// TIA Portal V20 export
DATA_BLOCK "ST_INPUT_Map_DB"   // DB102
{ S7_Optimized_Access := 'FALSE' }
// stored: AutoNumber false
   VAR
      "I0.0" { ExternalVisible := 'False'} : Bool := FALSE;   // I0.0
      "I0.1" { ExternalVisible := 'False'} : Bool := FALSE;   // I0.1
      "I0.2" { ExternalVisible := 'False'} : Bool := FALSE;   // I0.2
      "I0.3" { ExternalVisible := 'False'} : Bool := FALSE;   // I0.3
      "I0.4" { ExternalVisible := 'False'} : Bool := FALSE;   // I0.4
      "I0.5" { ExternalVisible := 'False'} : Bool := FALSE;   // I0.5
      "I0.6" { ExternalVisible := 'False'} : Bool := FALSE;   // I0.6
      "I0.7" { ExternalVisible := 'False'} : Bool := FALSE;   // I0.7
      "I1.0" { ExternalVisible := 'False'} : Bool := FALSE;   // I1.0
      "I1.1" { ExternalVisible := 'False'} : Bool := FALSE;   // I1.1
      "I1.2" { ExternalVisible := 'False'} : Bool := FALSE;   // I1.2
      "I1.3" { ExternalVisible := 'False'} : Bool := FALSE;   // I1.3
      "I1.4" { ExternalVisible := 'False'} : Bool := FALSE;   // I1.4
      "I1.5" { ExternalVisible := 'False'} : Bool := FALSE;   // I1.5
      "I1.6" { ExternalVisible := 'False'} : Bool := FALSE;   // I1.6
      "I1.7" { ExternalVisible := 'False'} : Bool := FALSE;   // I1.7
      "I2.0" { ExternalVisible := 'False'} : Bool := FALSE;   // I2.0
      "I2.1" { ExternalVisible := 'False'} : Bool := FALSE;   // I2.1
      "I2.2" { ExternalVisible := 'False'} : Bool := FALSE;   // I2.2
      "I2.3" { ExternalVisible := 'False'} : Bool := FALSE;   // I2.3
      "I2.4" { ExternalVisible := 'False'} : Bool := FALSE;   // I2.4
      "I2.5" { ExternalVisible := 'False'} : Bool := FALSE;   // I2.5
      "I2.6" { ExternalVisible := 'False'} : Bool := FALSE;   // I2.6
      "I2.7" { ExternalVisible := 'False'} : Bool := FALSE;   // I2.7
      "I3.0" { ExternalVisible := 'False'} : Bool := FALSE;   // I3.0
      "I3.1" { ExternalVisible := 'False'} : Bool := FALSE;   // I3.1
      "I3.2" { ExternalVisible := 'False'} : Bool := FALSE;   // I3.2
      "I3.3" { ExternalVisible := 'False'} : Bool := FALSE;   // I3.3
      "I3.4" { ExternalVisible := 'False'} : Bool := FALSE;   // I3.4
      "I3.5" { ExternalVisible := 'False'} : Bool := FALSE;   // I3.5
      "I3.6" { ExternalVisible := 'False'} : Bool := FALSE;   // I3.6
      "I3.7" { ExternalVisible := 'False'} : Bool := FALSE;   // I3.7
      "I4.0" { ExternalVisible := 'False'} : Bool := FALSE;   // I4.0
      "I4.1" { ExternalVisible := 'False'} : Bool := FALSE;   // I4.1
      "I4.2" { ExternalVisible := 'False'} : Bool := FALSE;   // I4.2
      "I4.3" { ExternalVisible := 'False'} : Bool := FALSE;   // I4.3
      "I4.4" { ExternalVisible := 'False'} : Bool := FALSE;   // I4.4
      "I4.5" { ExternalVisible := 'False'} : Bool := FALSE;   // I4.5
      "I4.6" { ExternalVisible := 'False'} : Bool := FALSE;   // I4.6
      "I4.7" { ExternalVisible := 'False'} : Bool := FALSE;   // I4.7
      "I5.0" { ExternalVisible := 'False'} : Bool := FALSE;   // I5.0
      "I5.1" { ExternalVisible := 'False'} : Bool := FALSE;   // I5.1
      "I5.2" { ExternalVisible := 'False'} : Bool := FALSE;   // I5.2
      "I5.3" { ExternalVisible := 'False'} : Bool := FALSE;   // I5.3
      "I5.4" { ExternalVisible := 'False'} : Bool := FALSE;   // I5.4
      "I5.5" { ExternalVisible := 'False'} : Bool := FALSE;   // I5.5
      "I5.6" { ExternalVisible := 'False'} : Bool := FALSE;   // I5.6
      "I5.7" { ExternalVisible := 'False'} : Bool := FALSE;   // I5.7
      "I6.0" { ExternalVisible := 'False'} : Bool := FALSE;   // I6.0
      "I6.1" { ExternalVisible := 'False'} : Bool := FALSE;   // I6.1
      "I6.2" { ExternalVisible := 'False'} : Bool := FALSE;   // I6.2
      "I6.3" { ExternalVisible := 'False'} : Bool := FALSE;   // I6.3
      "I6.4" { ExternalVisible := 'False'} : Bool := FALSE;   // I6.4
      "I6.5" { ExternalVisible := 'False'} : Bool := FALSE;   // I6.5
      "I6.6" { ExternalVisible := 'False'} : Bool := FALSE;   // I6.6
      "I6.7" { ExternalVisible := 'False'} : Bool := FALSE;   // I6.7
      "I7.0" { ExternalVisible := 'False'} : Bool := FALSE;   // I7.0
      "I7.1" { ExternalVisible := 'False'} : Bool := FALSE;   // I7.1
      "I7.2" { ExternalVisible := 'False'} : Bool := FALSE;   // I7.2
      "I7.3" { ExternalVisible := 'False'} : Bool := FALSE;   // I7.3
      "I7.4" { ExternalVisible := 'False'} : Bool := FALSE;   // I7.4
      "I7.5" { ExternalVisible := 'False'} : Bool := FALSE;   // I7.5
      "I7.6" { ExternalVisible := 'False'} : Bool := FALSE;   // I7.6
      "I7.7" { ExternalVisible := 'False'} : Bool := FALSE;   // I7.7
      "I8.0" { ExternalVisible := 'False'} : Bool := FALSE;   // I8.0
      "I8.1" { ExternalVisible := 'False'} : Bool := FALSE;   // I8.1
      "I8.2" { ExternalVisible := 'False'} : Bool := FALSE;   // I8.2
      "I8.3" { ExternalVisible := 'False'} : Bool := FALSE;   // I8.3
      "I8.4" { ExternalVisible := 'False'} : Bool := FALSE;   // I8.4
      "I8.5" { ExternalVisible := 'False'} : Bool := FALSE;   // I8.5
      "I8.6" { ExternalVisible := 'False'} : Bool := FALSE;   // I8.6
      "I8.7" { ExternalVisible := 'False'} : Bool := FALSE;   // I8.7
      "I9.0" { ExternalVisible := 'False'} : Bool := FALSE;   // I9.0
      "I9.1" { ExternalVisible := 'False'} : Bool := FALSE;   // I9.1
      "I9.2" { ExternalVisible := 'False'} : Bool := FALSE;   // I9.2
      "I9.3" { ExternalVisible := 'False'} : Bool := FALSE;   // I9.3
      "I9.4" { ExternalVisible := 'False'} : Bool := FALSE;   // I9.4
      "I9.5" { ExternalVisible := 'False'} : Bool := FALSE;   // I9.5
      "I9.6" { ExternalVisible := 'False'} : Bool := FALSE;   // I9.6
      "I9.7" { ExternalVisible := 'False'} : Bool := FALSE;   // I9.7
      F31 { ExternalVisible := 'False'} : Bool := FALSE;   // HMI供电反馈
      F32 { ExternalVisible := 'False'} : Bool := FALSE;   // ET200SP接口模块供电
      F33 { ExternalVisible := 'False'} : Bool := FALSE;   // 交换机供电反馈
      F34 { ExternalVisible := 'False'} : Bool := FALSE;   // FDI模块供电反馈
      F35 { ExternalVisible := 'False'} : Bool := FALSE;   // FDO模块供电反馈
      F36 { ExternalVisible := 'False'} : Bool := FALSE;   // DI模块供电反馈
      "I10.6" { ExternalVisible := 'False'} : Bool := FALSE;   // I10.6
      "I10.7" { ExternalVisible := 'False'} : Bool := FALSE;   // I10.7
      F37 { ExternalVisible := 'False'} : Bool := FALSE;   // DO模块¶供电反馈
      F38 { ExternalVisible := 'False'} : Bool := FALSE;   // 现场阀岛¶供电反馈
      F39 { ExternalVisible := 'False'} : Bool := FALSE;   // 现场IO模块¶供电反馈
      F40 { ExternalVisible := 'False'} : Bool := FALSE;   // 安全电源可控¶供电反馈
      F41 { ExternalVisible := 'False'} : Bool := FALSE;   // 安全门及¶上电控制电源¶供电反馈
      F42 { ExternalVisible := 'False'} : Bool := FALSE;   // 送纸伺服24V¶供电反馈
      F43 { ExternalVisible := 'False'} : Bool := FALSE;   // 滚纸伺服24V¶供电反馈
      F44 { ExternalVisible := 'False'} : Bool := FALSE;   // 分度伺服24V¶供电反馈
      F45 { ExternalVisible := 'False'} : Bool := FALSE;   // F45开关信号反馈
      F46 { ExternalVisible := 'False'} : Bool := FALSE;   // F46开关信号反馈
      F3 { ExternalVisible := 'False'} : Bool := FALSE;   // 送纸伺服¶供电反馈
      F47 { ExternalVisible := 'False'} : Bool := FALSE;   // 滚纸伺服¶供电反馈
      F48 { ExternalVisible := 'False'} : Bool := FALSE;   // 分度伺服¶供电反馈
      SB02 { ExternalVisible := 'False'} : Bool := FALSE;   // Lamp_Test
      SB03 { ExternalVisible := 'False'} : Bool := FALSE;   // Reset
      "I12.7" { ExternalVisible := 'False'} : Bool := FALSE;   // I12.7
      "GBS1-Y32" { ExternalVisible := 'False'} : Bool := FALSE;   // Safety Door 01 Closed
      "GBS2-Y32" { ExternalVisible := 'False'} : Bool := FALSE;   // Safety Door 02 Closed
      F4 { ExternalVisible := 'False'} : Bool := FALSE;   // 送纸伺服¶供电反馈
      F49 { ExternalVisible := 'False'} : Bool := FALSE;   // 滚纸伺服¶供电反馈
      F50 { ExternalVisible := 'False'} : Bool := FALSE;   // 分度伺服¶供电反馈
      "I13.5" { ExternalVisible := 'False'} : Bool := FALSE;   // I13.5
      "I13.6" { ExternalVisible := 'False'} : Bool := FALSE;   // I13.6
      "I13.7" { ExternalVisible := 'False'} : Bool := FALSE;   // I13.7
      "I14.0" { ExternalVisible := 'False'} : Bool := FALSE;   // I14.0
      "I14.1" { ExternalVisible := 'False'} : Bool := FALSE;   // I14.1
      "I14.2" { ExternalVisible := 'False'} : Bool := FALSE;   // I14.2
      "I14.3" { ExternalVisible := 'False'} : Bool := FALSE;   // I14.3
      "I14.4" { ExternalVisible := 'False'} : Bool := FALSE;   // I14.4
      "I14.5" { ExternalVisible := 'False'} : Bool := FALSE;   // I14.5
      "I14.6" { ExternalVisible := 'False'} : Bool := FALSE;   // I14.6
      "I14.7" { ExternalVisible := 'False'} : Bool := FALSE;   // I14.7
      "I15.0" { ExternalVisible := 'False'} : Bool := FALSE;   // I15.0
      "I15.1" { ExternalVisible := 'False'} : Bool := FALSE;   // I15.1
      "I15.2" { ExternalVisible := 'False'} : Bool := FALSE;   // I15.2
      "I15.3" { ExternalVisible := 'False'} : Bool := FALSE;   // I15.3
      "I15.4" { ExternalVisible := 'False'} : Bool := FALSE;   // I15.4
      "I15.5" { ExternalVisible := 'False'} : Bool := FALSE;   // I15.5
      "I15.6" { ExternalVisible := 'False'} : Bool := FALSE;   // I15.6
      "I15.7" { ExternalVisible := 'False'} : Bool := FALSE;   // I15.7
      "I16.0" { ExternalVisible := 'False'} : Bool := FALSE;   // I16.0
      "I16.1" { ExternalVisible := 'False'} : Bool := FALSE;   // I16.1
      "I16.2" { ExternalVisible := 'False'} : Bool := FALSE;   // I16.2
      "I16.3" { ExternalVisible := 'False'} : Bool := FALSE;   // I16.3
      "I16.4" { ExternalVisible := 'False'} : Bool := FALSE;   // I16.4
      "I16.5" { ExternalVisible := 'False'} : Bool := FALSE;   // I16.5
      "I16.6" { ExternalVisible := 'False'} : Bool := FALSE;   // I16.6
      "I16.7" { ExternalVisible := 'False'} : Bool := FALSE;   // I16.7
      "I17.0" { ExternalVisible := 'False'} : Bool := FALSE;   // I17.0
      "I17.1" { ExternalVisible := 'False'} : Bool := FALSE;   // I17.1
      "I17.2" { ExternalVisible := 'False'} : Bool := FALSE;   // I17.2
      "I17.3" { ExternalVisible := 'False'} : Bool := FALSE;   // I17.3
      "I17.4" { ExternalVisible := 'False'} : Bool := FALSE;   // I17.4
      "I17.5" { ExternalVisible := 'False'} : Bool := FALSE;   // I17.5
      "I17.6" { ExternalVisible := 'False'} : Bool := FALSE;   // I17.6
      "I17.7" { ExternalVisible := 'False'} : Bool := FALSE;   // I17.7
      "I18.0" { ExternalVisible := 'False'} : Bool := FALSE;   // I18.0
      "I18.1" { ExternalVisible := 'False'} : Bool := FALSE;   // I18.1
      "I18.2" { ExternalVisible := 'False'} : Bool := FALSE;   // I18.2
      "I18.3" { ExternalVisible := 'False'} : Bool := FALSE;   // I18.3
      "I18.4" { ExternalVisible := 'False'} : Bool := FALSE;   // I18.4
      "I18.5" { ExternalVisible := 'False'} : Bool := FALSE;   // I18.5
      "I18.6" { ExternalVisible := 'False'} : Bool := FALSE;   // I18.6
      "I18.7" { ExternalVisible := 'False'} : Bool := FALSE;   // I18.7
      "I19.0" { ExternalVisible := 'False'} : Bool := FALSE;   // I19.0
      "I19.1" { ExternalVisible := 'False'} : Bool := FALSE;   // I19.1
      "I19.2" { ExternalVisible := 'False'} : Bool := FALSE;   // I19.2
      "I19.3" { ExternalVisible := 'False'} : Bool := FALSE;   // I19.3
      "I19.4" { ExternalVisible := 'False'} : Bool := FALSE;   // I19.4
      "I19.5" { ExternalVisible := 'False'} : Bool := FALSE;   // I19.5
      "I19.6" { ExternalVisible := 'False'} : Bool := FALSE;   // I19.6
      "I19.7" { ExternalVisible := 'False'} : Bool := FALSE;   // I19.7
      "I20.0" { ExternalVisible := 'False'} : Bool := FALSE;   // I20.0
      "I20.1" { ExternalVisible := 'False'} : Bool := FALSE;   // I20.1
      "I20.2" { ExternalVisible := 'False'} : Bool := FALSE;   // I20.2
      "I20.3" { ExternalVisible := 'False'} : Bool := FALSE;   // I20.3
      "I20.4" { ExternalVisible := 'False'} : Bool := FALSE;   // I20.4
      "I20.5" { ExternalVisible := 'False'} : Bool := FALSE;   // I20.5
      "I20.6" { ExternalVisible := 'False'} : Bool := FALSE;   // I20.6
      "I20.7" { ExternalVisible := 'False'} : Bool := FALSE;   // I20.7
      "I21.0" { ExternalVisible := 'False'} : Bool := FALSE;   // I21.0
      "I21.1" { ExternalVisible := 'False'} : Bool := FALSE;   // I21.1
      "I21.2" { ExternalVisible := 'False'} : Bool := FALSE;   // I21.2
      "I21.3" { ExternalVisible := 'False'} : Bool := FALSE;   // I21.3
      "I21.4" { ExternalVisible := 'False'} : Bool := FALSE;   // I21.4
      "I21.5" { ExternalVisible := 'False'} : Bool := FALSE;   // I21.5
      "I21.6" { ExternalVisible := 'False'} : Bool := FALSE;   // I21.6
      "I21.7" { ExternalVisible := 'False'} : Bool := FALSE;   // I21.7
      "I22.0" { ExternalVisible := 'False'} : Bool := FALSE;   // I22.0
      "I22.1" { ExternalVisible := 'False'} : Bool := FALSE;   // I22.1
      "I22.2" { ExternalVisible := 'False'} : Bool := FALSE;   // I22.2
      "I22.3" { ExternalVisible := 'False'} : Bool := FALSE;   // I22.3
      "I22.4" { ExternalVisible := 'False'} : Bool := FALSE;   // I22.4
      "I22.5" { ExternalVisible := 'False'} : Bool := FALSE;   // I22.5
      "I22.6" { ExternalVisible := 'False'} : Bool := FALSE;   // I22.6
      "I22.7" { ExternalVisible := 'False'} : Bool := FALSE;   // I22.7
      "I23.0" { ExternalVisible := 'False'} : Bool := FALSE;   // I23.0
      "I23.1" { ExternalVisible := 'False'} : Bool := FALSE;   // I23.1
      "I23.2" { ExternalVisible := 'False'} : Bool := FALSE;   // I23.2
      "I23.3" { ExternalVisible := 'False'} : Bool := FALSE;   // I23.3
      "I23.4" { ExternalVisible := 'False'} : Bool := FALSE;   // I23.4
      "I23.5" { ExternalVisible := 'False'} : Bool := FALSE;   // I23.5
      "I23.6" { ExternalVisible := 'False'} : Bool := FALSE;   // I23.6
      "I23.7" { ExternalVisible := 'False'} : Bool := FALSE;   // I23.7
      "I24.0" { ExternalVisible := 'False'} : Bool := FALSE;   // I24.0
      "I24.1" { ExternalVisible := 'False'} : Bool := FALSE;   // I24.1
      "I24.2" { ExternalVisible := 'False'} : Bool := FALSE;   // I24.2
      "I24.3" { ExternalVisible := 'False'} : Bool := FALSE;   // I24.3
      "I24.4" { ExternalVisible := 'False'} : Bool := FALSE;   // I24.4
      "I24.5" { ExternalVisible := 'False'} : Bool := FALSE;   // I24.5
      "I24.6" { ExternalVisible := 'False'} : Bool := FALSE;   // I24.6
      "I24.7" { ExternalVisible := 'False'} : Bool := FALSE;   // I24.7
      "I25.0" { ExternalVisible := 'False'} : Bool := FALSE;   // I25.0
      "I25.1" { ExternalVisible := 'False'} : Bool := FALSE;   // I25.1
      "I25.2" { ExternalVisible := 'False'} : Bool := FALSE;   // I25.2
      "I25.3" { ExternalVisible := 'False'} : Bool := FALSE;   // I25.3
      "I25.4" { ExternalVisible := 'False'} : Bool := FALSE;   // I25.4
      "I25.5" { ExternalVisible := 'False'} : Bool := FALSE;   // I25.5
      "I25.6" { ExternalVisible := 'False'} : Bool := FALSE;   // I25.6
      "I25.7" { ExternalVisible := 'False'} : Bool := FALSE;   // I25.7
      "I26.0" { ExternalVisible := 'False'} : Bool := FALSE;   // I26.0
      "I26.1" { ExternalVisible := 'False'} : Bool := FALSE;   // I26.1
      "I26.2" { ExternalVisible := 'False'} : Bool := FALSE;   // I26.2
      "I26.3" { ExternalVisible := 'False'} : Bool := FALSE;   // I26.3
      "I26.4" { ExternalVisible := 'False'} : Bool := FALSE;   // I26.4
      "I26.5" { ExternalVisible := 'False'} : Bool := FALSE;   // I26.5
      "I26.6" { ExternalVisible := 'False'} : Bool := FALSE;   // I26.6
      "I26.7" { ExternalVisible := 'False'} : Bool := FALSE;   // I26.7
      "I27.0" { ExternalVisible := 'False'} : Bool := FALSE;   // I27.0
      "I27.1" { ExternalVisible := 'False'} : Bool := FALSE;   // I27.1
      "I27.2" { ExternalVisible := 'False'} : Bool := FALSE;   // I27.2
      "I27.3" { ExternalVisible := 'False'} : Bool := FALSE;   // I27.3
      "I27.4" { ExternalVisible := 'False'} : Bool := FALSE;   // I27.4
      "I27.5" { ExternalVisible := 'False'} : Bool := FALSE;   // I27.5
      "I27.6" { ExternalVisible := 'False'} : Bool := FALSE;   // I27.6
      "I27.7" { ExternalVisible := 'False'} : Bool := FALSE;   // I27.7
      "I28.0" { ExternalVisible := 'False'} : Bool := FALSE;   // I28.0
      "I28.1" { ExternalVisible := 'False'} : Bool := FALSE;   // I28.1
      "I28.2" { ExternalVisible := 'False'} : Bool := FALSE;   // I28.2
      "I28.3" { ExternalVisible := 'False'} : Bool := FALSE;   // I28.3
      "I28.4" { ExternalVisible := 'False'} : Bool := FALSE;   // I28.4
      "I28.5" { ExternalVisible := 'False'} : Bool := FALSE;   // I28.5
      "I28.6" { ExternalVisible := 'False'} : Bool := FALSE;   // I28.6
      "I28.7" { ExternalVisible := 'False'} : Bool := FALSE;   // I28.7
      "I29.0" { ExternalVisible := 'False'} : Bool := FALSE;   // I29.0
      "I29.1" { ExternalVisible := 'False'} : Bool := FALSE;   // I29.1
      "I29.2" { ExternalVisible := 'False'} : Bool := FALSE;   // I29.2
      "I29.3" { ExternalVisible := 'False'} : Bool := FALSE;   // I29.3
      "I29.4" { ExternalVisible := 'False'} : Bool := FALSE;   // I29.4
      "I29.5" { ExternalVisible := 'False'} : Bool := FALSE;   // I29.5
      "I29.6" { ExternalVisible := 'False'} : Bool := FALSE;   // I29.6
      "I29.7" { ExternalVisible := 'False'} : Bool := FALSE;   // I29.7
      "I30.0" { ExternalVisible := 'False'} : Bool := FALSE;   // I30.0
      "I30.1" { ExternalVisible := 'False'} : Bool := FALSE;   // I30.1
      "I30.2" { ExternalVisible := 'False'} : Bool := FALSE;   // I30.2
      "I30.3" { ExternalVisible := 'False'} : Bool := FALSE;   // I30.3
      "I30.4" { ExternalVisible := 'False'} : Bool := FALSE;   // I30.4
      "I30.5" { ExternalVisible := 'False'} : Bool := FALSE;   // I30.5
      "I30.6" { ExternalVisible := 'False'} : Bool := FALSE;   // I30.6
      "I30.7" { ExternalVisible := 'False'} : Bool := FALSE;   // I30.7
      "I31.0" { ExternalVisible := 'False'} : Bool := FALSE;   // I31.0
      "I31.1" { ExternalVisible := 'False'} : Bool := FALSE;   // I31.1
      "I31.2" { ExternalVisible := 'False'} : Bool := FALSE;   // I31.2
      "I31.3" { ExternalVisible := 'False'} : Bool := FALSE;   // I31.3
      "I31.4" { ExternalVisible := 'False'} : Bool := FALSE;   // I31.4
      "I31.5" { ExternalVisible := 'False'} : Bool := FALSE;   // I31.5
      "I31.6" { ExternalVisible := 'False'} : Bool := FALSE;   // I31.6
      "I31.7" { ExternalVisible := 'False'} : Bool := FALSE;   // I31.7
      "I32.0" { ExternalVisible := 'False'} : Bool := FALSE;   // I32.0
      "I32.1" { ExternalVisible := 'False'} : Bool := FALSE;   // I32.1
      "I32.2" { ExternalVisible := 'False'} : Bool := FALSE;   // I32.2
      "I32.3" { ExternalVisible := 'False'} : Bool := FALSE;   // I32.3
      "I32.4" { ExternalVisible := 'False'} : Bool := FALSE;   // I32.4
      "I32.5" { ExternalVisible := 'False'} : Bool := FALSE;   // I32.5
      "I32.6" { ExternalVisible := 'False'} : Bool := FALSE;   // I32.6
      "I32.7" { ExternalVisible := 'False'} : Bool := FALSE;   // I32.7
      "I33.0" { ExternalVisible := 'False'} : Bool := FALSE;   // I33.0
      "I33.1" { ExternalVisible := 'False'} : Bool := FALSE;   // I33.1
      "I33.2" { ExternalVisible := 'False'} : Bool := FALSE;   // I33.2
      "I33.3" { ExternalVisible := 'False'} : Bool := FALSE;   // I33.3
      "I33.4" { ExternalVisible := 'False'} : Bool := FALSE;   // I33.4
      "I33.5" { ExternalVisible := 'False'} : Bool := FALSE;   // I33.5
      "I33.6" { ExternalVisible := 'False'} : Bool := FALSE;   // I33.6
      "I33.7" { ExternalVisible := 'False'} : Bool := FALSE;   // I33.7
      "I34.0" { ExternalVisible := 'False'} : Bool := FALSE;   // I34.0
      "I34.1" { ExternalVisible := 'False'} : Bool := FALSE;   // I34.1
      "I34.2" { ExternalVisible := 'False'} : Bool := FALSE;   // I34.2
      "I34.3" { ExternalVisible := 'False'} : Bool := FALSE;   // I34.3
      "I34.4" { ExternalVisible := 'False'} : Bool := FALSE;   // I34.4
      "I34.5" { ExternalVisible := 'False'} : Bool := FALSE;   // I34.5
      "I34.6" { ExternalVisible := 'False'} : Bool := FALSE;   // I34.6
      "I34.7" { ExternalVisible := 'False'} : Bool := FALSE;   // I34.7
      "I35.0" { ExternalVisible := 'False'} : Bool := FALSE;   // I35.0
      "I35.1" { ExternalVisible := 'False'} : Bool := FALSE;   // I35.1
      "I35.2" { ExternalVisible := 'False'} : Bool := FALSE;   // I35.2
      "I35.3" { ExternalVisible := 'False'} : Bool := FALSE;   // I35.3
      "I35.4" { ExternalVisible := 'False'} : Bool := FALSE;   // I35.4
      "I35.5" { ExternalVisible := 'False'} : Bool := FALSE;   // I35.5
      "I35.6" { ExternalVisible := 'False'} : Bool := FALSE;   // I35.6
      "I35.7" { ExternalVisible := 'False'} : Bool := FALSE;   // I35.7
      "I36.0" { ExternalVisible := 'False'} : Bool := FALSE;   // I36.0
      "I36.1" { ExternalVisible := 'False'} : Bool := FALSE;   // I36.1
      "I36.2" { ExternalVisible := 'False'} : Bool := FALSE;   // I36.2
      "I36.3" { ExternalVisible := 'False'} : Bool := FALSE;   // I36.3
      "I36.4" { ExternalVisible := 'False'} : Bool := FALSE;   // I36.4
      "I36.5" { ExternalVisible := 'False'} : Bool := FALSE;   // I36.5
      "I36.6" { ExternalVisible := 'False'} : Bool := FALSE;   // I36.6
      "I36.7" { ExternalVisible := 'False'} : Bool := FALSE;   // I36.7
      "I37.0" { ExternalVisible := 'False'} : Bool := FALSE;   // I37.0
      "I37.1" { ExternalVisible := 'False'} : Bool := FALSE;   // I37.1
      "I37.2" { ExternalVisible := 'False'} : Bool := FALSE;   // I37.2
      "I37.3" { ExternalVisible := 'False'} : Bool := FALSE;   // I37.3
      "I37.4" { ExternalVisible := 'False'} : Bool := FALSE;   // I37.4
      "I37.5" { ExternalVisible := 'False'} : Bool := FALSE;   // I37.5
      "I37.6" { ExternalVisible := 'False'} : Bool := FALSE;   // I37.6
      "I37.7" { ExternalVisible := 'False'} : Bool := FALSE;   // I37.7
      "I38.0" { ExternalVisible := 'False'} : Bool := FALSE;   // I38.0
      "I38.1" { ExternalVisible := 'False'} : Bool := FALSE;   // I38.1
      "I38.2" { ExternalVisible := 'False'} : Bool := FALSE;   // I38.2
      "I38.3" { ExternalVisible := 'False'} : Bool := FALSE;   // I38.3
      "I38.4" { ExternalVisible := 'False'} : Bool := FALSE;   // I38.4
      "I38.5" { ExternalVisible := 'False'} : Bool := FALSE;   // I38.5
      "I38.6" { ExternalVisible := 'False'} : Bool := FALSE;   // I38.6
      "I38.7" { ExternalVisible := 'False'} : Bool := FALSE;   // I38.7
      "I39.0" { ExternalVisible := 'False'} : Bool := FALSE;   // I39.0
      "I39.1" { ExternalVisible := 'False'} : Bool := FALSE;   // I39.1
      "I39.2" { ExternalVisible := 'False'} : Bool := FALSE;   // I39.2
      "I39.3" { ExternalVisible := 'False'} : Bool := FALSE;   // I39.3
      "I39.4" { ExternalVisible := 'False'} : Bool := FALSE;   // I39.4
      "I39.5" { ExternalVisible := 'False'} : Bool := FALSE;   // I39.5
      "I39.6" { ExternalVisible := 'False'} : Bool := FALSE;   // I39.6
      "I39.7" { ExternalVisible := 'False'} : Bool := FALSE;   // I39.7
      "I40.0" { ExternalVisible := 'False'} : Bool := FALSE;   // I40.0
      "I40.1" { ExternalVisible := 'False'} : Bool := FALSE;   // I40.1
      "I40.2" { ExternalVisible := 'False'} : Bool := FALSE;   // I40.2
      "I40.3" { ExternalVisible := 'False'} : Bool := FALSE;   // I40.3
      "I40.4" { ExternalVisible := 'False'} : Bool := FALSE;   // I40.4
      "I40.5" { ExternalVisible := 'False'} : Bool := FALSE;   // I40.5
      "I40.6" { ExternalVisible := 'False'} : Bool := FALSE;   // I40.6
      "I40.7" { ExternalVisible := 'False'} : Bool := FALSE;   // I40.7
      "I41.0" { ExternalVisible := 'False'} : Bool := FALSE;   // I41.0
      "I41.1" { ExternalVisible := 'False'} : Bool := FALSE;   // I41.1
      "I41.2" { ExternalVisible := 'False'} : Bool := FALSE;   // I41.2
      "I41.3" { ExternalVisible := 'False'} : Bool := FALSE;   // I41.3
      "I41.4" { ExternalVisible := 'False'} : Bool := FALSE;   // I41.4
      "I41.5" { ExternalVisible := 'False'} : Bool := FALSE;   // I41.5
      "I41.6" { ExternalVisible := 'False'} : Bool := FALSE;   // I41.6
      "I41.7" { ExternalVisible := 'False'} : Bool := FALSE;   // I41.7
      "I42.0" { ExternalVisible := 'False'} : Bool := FALSE;   // I42.0
      "I42.1" { ExternalVisible := 'False'} : Bool := FALSE;   // I42.1
      "I42.2" { ExternalVisible := 'False'} : Bool := FALSE;   // I42.2
      "I42.3" { ExternalVisible := 'False'} : Bool := FALSE;   // I42.3
      "I42.4" { ExternalVisible := 'False'} : Bool := FALSE;   // I42.4
      "I42.5" { ExternalVisible := 'False'} : Bool := FALSE;   // I42.5
      "I42.6" { ExternalVisible := 'False'} : Bool := FALSE;   // I42.6
      "I42.7" { ExternalVisible := 'False'} : Bool := FALSE;   // I42.7
      "I43.0" { ExternalVisible := 'False'} : Bool := FALSE;   // I43.0
      "I43.1" { ExternalVisible := 'False'} : Bool := FALSE;   // I43.1
      "I43.2" { ExternalVisible := 'False'} : Bool := FALSE;   // I43.2
      "I43.3" { ExternalVisible := 'False'} : Bool := FALSE;   // I43.3
      "I43.4" { ExternalVisible := 'False'} : Bool := FALSE;   // I43.4
      "I43.5" { ExternalVisible := 'False'} : Bool := FALSE;   // I43.5
      "I43.6" { ExternalVisible := 'False'} : Bool := FALSE;   // I43.6
      "I43.7" { ExternalVisible := 'False'} : Bool := FALSE;   // I43.7
      "I44.0" { ExternalVisible := 'False'} : Bool := FALSE;   // I44.0
      "I44.1" { ExternalVisible := 'False'} : Bool := FALSE;   // I44.1
      "I44.2" { ExternalVisible := 'False'} : Bool := FALSE;   // I44.2
      "I44.3" { ExternalVisible := 'False'} : Bool := FALSE;   // I44.3
      "I44.4" { ExternalVisible := 'False'} : Bool := FALSE;   // I44.4
      "I44.5" { ExternalVisible := 'False'} : Bool := FALSE;   // I44.5
      "I44.6" { ExternalVisible := 'False'} : Bool := FALSE;   // I44.6
      "I44.7" { ExternalVisible := 'False'} : Bool := FALSE;   // I44.7
      "I45.0" { ExternalVisible := 'False'} : Bool := FALSE;   // I45.0
      "I45.1" { ExternalVisible := 'False'} : Bool := FALSE;   // I45.1
      "I45.2" { ExternalVisible := 'False'} : Bool := FALSE;   // I45.2
      "I45.3" { ExternalVisible := 'False'} : Bool := FALSE;   // I45.3
      "I45.4" { ExternalVisible := 'False'} : Bool := FALSE;   // I45.4
      "I45.5" { ExternalVisible := 'False'} : Bool := FALSE;   // I45.5
      "I45.6" { ExternalVisible := 'False'} : Bool := FALSE;   // I45.6
      "I45.7" { ExternalVisible := 'False'} : Bool := FALSE;   // I45.7
      "I46.0" { ExternalVisible := 'False'} : Bool := FALSE;   // I46.0
      "I46.1" { ExternalVisible := 'False'} : Bool := FALSE;   // I46.1
      "I46.2" { ExternalVisible := 'False'} : Bool := FALSE;   // I46.2
      "I46.3" { ExternalVisible := 'False'} : Bool := FALSE;   // I46.3
      "I46.4" { ExternalVisible := 'False'} : Bool := FALSE;   // I46.4
      "I46.5" { ExternalVisible := 'False'} : Bool := FALSE;   // I46.5
      "I46.6" { ExternalVisible := 'False'} : Bool := FALSE;   // I46.6
      "I46.7" { ExternalVisible := 'False'} : Bool := FALSE;   // I46.7
      "I47.0" { ExternalVisible := 'False'} : Bool := FALSE;   // I47.0
      "I47.1" { ExternalVisible := 'False'} : Bool := FALSE;   // I47.1
      "I47.2" { ExternalVisible := 'False'} : Bool := FALSE;   // I47.2
      "I47.3" { ExternalVisible := 'False'} : Bool := FALSE;   // I47.3
      "I47.4" { ExternalVisible := 'False'} : Bool := FALSE;   // I47.4
      "I47.5" { ExternalVisible := 'False'} : Bool := FALSE;   // I47.5
      "I47.6" { ExternalVisible := 'False'} : Bool := FALSE;   // I47.6
      "I47.7" { ExternalVisible := 'False'} : Bool := FALSE;   // I47.7
      "I48.0" { ExternalVisible := 'False'} : Bool := FALSE;   // I48.0
      "I48.1" { ExternalVisible := 'False'} : Bool := FALSE;   // I48.1
      "I48.2" { ExternalVisible := 'False'} : Bool := FALSE;   // I48.2
      "I48.3" { ExternalVisible := 'False'} : Bool := FALSE;   // I48.3
      "I48.4" { ExternalVisible := 'False'} : Bool := FALSE;   // I48.4
      "I48.5" { ExternalVisible := 'False'} : Bool := FALSE;   // I48.5
      "I48.6" { ExternalVisible := 'False'} : Bool := FALSE;   // I48.6
      "I48.7" { ExternalVisible := 'False'} : Bool := FALSE;   // I48.7
      "I49.0" { ExternalVisible := 'False'} : Bool := FALSE;   // I49.0
      "I49.1" { ExternalVisible := 'False'} : Bool := FALSE;   // I49.1
      "I49.2" { ExternalVisible := 'False'} : Bool := FALSE;   // I49.2
      "I49.3" { ExternalVisible := 'False'} : Bool := FALSE;   // I49.3
      "I49.4" { ExternalVisible := 'False'} : Bool := FALSE;   // I49.4
      "I49.5" { ExternalVisible := 'False'} : Bool := FALSE;   // I49.5
      "I49.6" { ExternalVisible := 'False'} : Bool := FALSE;   // I49.6
      "I49.7" { ExternalVisible := 'False'} : Bool := FALSE;   // I49.7
      "I50.0" { ExternalVisible := 'False'} : Bool := FALSE;   // I50.0
      "I50.1" { ExternalVisible := 'False'} : Bool := FALSE;   // I50.1
      "I50.2" { ExternalVisible := 'False'} : Bool := FALSE;   // I50.2
      "I50.3" { ExternalVisible := 'False'} : Bool := FALSE;   // I50.3
      "I50.4" { ExternalVisible := 'False'} : Bool := FALSE;   // I50.4
      "I50.5" { ExternalVisible := 'False'} : Bool := FALSE;   // I50.5
      "I50.6" { ExternalVisible := 'False'} : Bool := FALSE;   // I50.6
      "I50.7" { ExternalVisible := 'False'} : Bool := FALSE;   // I50.7
      "I51.0" { ExternalVisible := 'False'} : Bool := FALSE;   // I51.0
      "I51.1" { ExternalVisible := 'False'} : Bool := FALSE;   // I51.1
      "I51.2" { ExternalVisible := 'False'} : Bool := FALSE;   // I51.2
      "I51.3" { ExternalVisible := 'False'} : Bool := FALSE;   // I51.3
      "I51.4" { ExternalVisible := 'False'} : Bool := FALSE;   // I51.4
      "I51.5" { ExternalVisible := 'False'} : Bool := FALSE;   // I51.5
      "I51.6" { ExternalVisible := 'False'} : Bool := FALSE;   // I51.6
      "I51.7" { ExternalVisible := 'False'} : Bool := FALSE;   // I51.7
      "I52.0" { ExternalVisible := 'False'} : Bool := FALSE;   // I52.0
      "I52.1" { ExternalVisible := 'False'} : Bool := FALSE;   // I52.1
      "I52.2" { ExternalVisible := 'False'} : Bool := FALSE;   // I52.2
      "I52.3" { ExternalVisible := 'False'} : Bool := FALSE;   // I52.3
      "I52.4" { ExternalVisible := 'False'} : Bool := FALSE;   // I52.4
      "I52.5" { ExternalVisible := 'False'} : Bool := FALSE;   // I52.5
      "I52.6" { ExternalVisible := 'False'} : Bool := FALSE;   // I52.6
      "I52.7" { ExternalVisible := 'False'} : Bool := FALSE;   // I52.7
      "I53.0" { ExternalVisible := 'False'} : Bool := FALSE;   // I53.0
      "I53.1" { ExternalVisible := 'False'} : Bool := FALSE;   // I53.1
      "I53.2" { ExternalVisible := 'False'} : Bool := FALSE;   // I53.2
      "I53.3" { ExternalVisible := 'False'} : Bool := FALSE;   // I53.3
      "I53.4" { ExternalVisible := 'False'} : Bool := FALSE;   // I53.4
      "I53.5" { ExternalVisible := 'False'} : Bool := FALSE;   // I53.5
      "I53.6" { ExternalVisible := 'False'} : Bool := FALSE;   // I53.6
      "I53.7" { ExternalVisible := 'False'} : Bool := FALSE;   // I53.7
      "I54.0" { ExternalVisible := 'False'} : Bool := FALSE;   // I54.0
      "I54.1" { ExternalVisible := 'False'} : Bool := FALSE;   // I54.1
      "I54.2" { ExternalVisible := 'False'} : Bool := FALSE;   // I54.2
      "I54.3" { ExternalVisible := 'False'} : Bool := FALSE;   // I54.3
      "I54.4" { ExternalVisible := 'False'} : Bool := FALSE;   // I54.4
      "I54.5" { ExternalVisible := 'False'} : Bool := FALSE;   // I54.5
      "I54.6" { ExternalVisible := 'False'} : Bool := FALSE;   // I54.6
      "I54.7" { ExternalVisible := 'False'} : Bool := FALSE;   // I54.7
      "I55.0" { ExternalVisible := 'False'} : Bool := FALSE;   // I55.0
      "I55.1" { ExternalVisible := 'False'} : Bool := FALSE;   // I55.1
      "I55.2" { ExternalVisible := 'False'} : Bool := FALSE;   // I55.2
      "I55.3" { ExternalVisible := 'False'} : Bool := FALSE;   // I55.3
      "I55.4" { ExternalVisible := 'False'} : Bool := FALSE;   // I55.4
      "I55.5" { ExternalVisible := 'False'} : Bool := FALSE;   // I55.5
      "I55.6" { ExternalVisible := 'False'} : Bool := FALSE;   // I55.6
      "I55.7" { ExternalVisible := 'False'} : Bool := FALSE;   // I55.7
      "I56.0" { ExternalVisible := 'False'} : Bool := FALSE;   // I56.0
      "I56.1" { ExternalVisible := 'False'} : Bool := FALSE;   // I56.1
      "I56.2" { ExternalVisible := 'False'} : Bool := FALSE;   // I56.2
      "I56.3" { ExternalVisible := 'False'} : Bool := FALSE;   // I56.3
      "I56.4" { ExternalVisible := 'False'} : Bool := FALSE;   // I56.4
      "I56.5" { ExternalVisible := 'False'} : Bool := FALSE;   // I56.5
      "I56.6" { ExternalVisible := 'False'} : Bool := FALSE;   // I56.6
      "I56.7" { ExternalVisible := 'False'} : Bool := FALSE;   // I56.7
      "I57.0" { ExternalVisible := 'False'} : Bool := FALSE;   // I57.0
      "I57.1" { ExternalVisible := 'False'} : Bool := FALSE;   // I57.1
      "I57.2" { ExternalVisible := 'False'} : Bool := FALSE;   // I57.2
      "I57.3" { ExternalVisible := 'False'} : Bool := FALSE;   // I57.3
      "I57.4" { ExternalVisible := 'False'} : Bool := FALSE;   // I57.4
      "I57.5" { ExternalVisible := 'False'} : Bool := FALSE;   // I57.5
      "I57.6" { ExternalVisible := 'False'} : Bool := FALSE;   // I57.6
      "I57.7" { ExternalVisible := 'False'} : Bool := FALSE;   // I57.7
      "I58.0" { ExternalVisible := 'False'} : Bool := FALSE;   // I58.0
      "I58.1" { ExternalVisible := 'False'} : Bool := FALSE;   // I58.1
      "I58.2" { ExternalVisible := 'False'} : Bool := FALSE;   // I58.2
      "I58.3" { ExternalVisible := 'False'} : Bool := FALSE;   // I58.3
      "I58.4" { ExternalVisible := 'False'} : Bool := FALSE;   // I58.4
      "I58.5" { ExternalVisible := 'False'} : Bool := FALSE;   // I58.5
      "I58.6" { ExternalVisible := 'False'} : Bool := FALSE;   // I58.6
      "I58.7" { ExternalVisible := 'False'} : Bool := FALSE;   // I58.7
      "I59.0" { ExternalVisible := 'False'} : Bool := FALSE;   // I59.0
      "I59.1" { ExternalVisible := 'False'} : Bool := FALSE;   // I59.1
      "I59.2" { ExternalVisible := 'False'} : Bool := FALSE;   // I59.2
      "I59.3" { ExternalVisible := 'False'} : Bool := FALSE;   // I59.3
      "I59.4" { ExternalVisible := 'False'} : Bool := FALSE;   // I59.4
      "I59.5" { ExternalVisible := 'False'} : Bool := FALSE;   // I59.5
      "I59.6" { ExternalVisible := 'False'} : Bool := FALSE;   // I59.6
      "I59.7" { ExternalVisible := 'False'} : Bool := FALSE;   // I59.7
      "I60.0" { ExternalVisible := 'False'} : Bool := FALSE;   // I60.0
      "I60.1" { ExternalVisible := 'False'} : Bool := FALSE;   // I60.1
      "I60.2" { ExternalVisible := 'False'} : Bool := FALSE;   // I60.2
      "I60.3" { ExternalVisible := 'False'} : Bool := FALSE;   // I60.3
      "I60.4" { ExternalVisible := 'False'} : Bool := FALSE;   // I60.4
      "I60.5" { ExternalVisible := 'False'} : Bool := FALSE;   // I60.5
      "I60.6" { ExternalVisible := 'False'} : Bool := FALSE;   // I60.6
      "I60.7" { ExternalVisible := 'False'} : Bool := FALSE;   // I60.7
      "I61.0" { ExternalVisible := 'False'} : Bool := FALSE;   // I61.0
      "I61.1" { ExternalVisible := 'False'} : Bool := FALSE;   // I61.1
      "I61.2" { ExternalVisible := 'False'} : Bool := FALSE;   // I61.2
      "I61.3" { ExternalVisible := 'False'} : Bool := FALSE;   // I61.3
      "I61.4" { ExternalVisible := 'False'} : Bool := FALSE;   // I61.4
      "I61.5" { ExternalVisible := 'False'} : Bool := FALSE;   // I61.5
      "I61.6" { ExternalVisible := 'False'} : Bool := FALSE;   // I61.6
      "I61.7" { ExternalVisible := 'False'} : Bool := FALSE;   // I61.7
      "I62.0" { ExternalVisible := 'False'} : Bool := FALSE;   // I62.0
      "I62.1" { ExternalVisible := 'False'} : Bool := FALSE;   // I62.1
      "I62.2" { ExternalVisible := 'False'} : Bool := FALSE;   // I62.2
      "I62.3" { ExternalVisible := 'False'} : Bool := FALSE;   // I62.3
      "I62.4" { ExternalVisible := 'False'} : Bool := FALSE;   // I62.4
      "I62.5" { ExternalVisible := 'False'} : Bool := FALSE;   // I62.5
      "I62.6" { ExternalVisible := 'False'} : Bool := FALSE;   // I62.6
      "I62.7" { ExternalVisible := 'False'} : Bool := FALSE;   // I62.7
      "I63.0" { ExternalVisible := 'False'} : Bool := FALSE;   // I63.0
      "I63.1" { ExternalVisible := 'False'} : Bool := FALSE;   // I63.1
      "I63.2" { ExternalVisible := 'False'} : Bool := FALSE;   // I63.2
      "I63.3" { ExternalVisible := 'False'} : Bool := FALSE;   // I63.3
      "I63.4" { ExternalVisible := 'False'} : Bool := FALSE;   // I63.4
      "I63.5" { ExternalVisible := 'False'} : Bool := FALSE;   // I63.5
      "I63.6" { ExternalVisible := 'False'} : Bool := FALSE;   // I63.6
      "I63.7" { ExternalVisible := 'False'} : Bool := FALSE;   // I63.7
      "I64.0" { ExternalVisible := 'False'} : Bool := FALSE;   // I64.0
      "I64.1" { ExternalVisible := 'False'} : Bool := FALSE;   // I64.1
      "I64.2" { ExternalVisible := 'False'} : Bool := FALSE;   // I64.2
      "I64.3" { ExternalVisible := 'False'} : Bool := FALSE;   // I64.3
      "I64.4" { ExternalVisible := 'False'} : Bool := FALSE;   // I64.4
      "I64.5" { ExternalVisible := 'False'} : Bool := FALSE;   // I64.5
      "I64.6" { ExternalVisible := 'False'} : Bool := FALSE;   // I64.6
      "I64.7" { ExternalVisible := 'False'} : Bool := FALSE;   // I64.7
      "I65.0" { ExternalVisible := 'False'} : Bool := FALSE;   // I65.0
      "I65.1" { ExternalVisible := 'False'} : Bool := FALSE;   // I65.1
      "I65.2" { ExternalVisible := 'False'} : Bool := FALSE;   // I65.2
      "I65.3" { ExternalVisible := 'False'} : Bool := FALSE;   // I65.3
      "I65.4" { ExternalVisible := 'False'} : Bool := FALSE;   // I65.4
      "I65.5" { ExternalVisible := 'False'} : Bool := FALSE;   // I65.5
      "I65.6" { ExternalVisible := 'False'} : Bool := FALSE;   // I65.6
      "I65.7" { ExternalVisible := 'False'} : Bool := FALSE;   // I65.7
      "I66.0" { ExternalVisible := 'False'} : Bool := FALSE;   // I66.0
      "I66.1" { ExternalVisible := 'False'} : Bool := FALSE;   // I66.1
      "I66.2" { ExternalVisible := 'False'} : Bool := FALSE;   // I66.2
      "I66.3" { ExternalVisible := 'False'} : Bool := FALSE;   // I66.3
      "I66.4" { ExternalVisible := 'False'} : Bool := FALSE;   // I66.4
      "I66.5" { ExternalVisible := 'False'} : Bool := FALSE;   // I66.5
      "I66.6" { ExternalVisible := 'False'} : Bool := FALSE;   // I66.6
      "I66.7" { ExternalVisible := 'False'} : Bool := FALSE;   // I66.7
      "I67.0" { ExternalVisible := 'False'} : Bool := FALSE;   // I67.0
      "I67.1" { ExternalVisible := 'False'} : Bool := FALSE;   // I67.1
      "I67.2" { ExternalVisible := 'False'} : Bool := FALSE;   // I67.2
      "I67.3" { ExternalVisible := 'False'} : Bool := FALSE;   // I67.3
      "I67.4" { ExternalVisible := 'False'} : Bool := FALSE;   // I67.4
      "I67.5" { ExternalVisible := 'False'} : Bool := FALSE;   // I67.5
      "I67.6" { ExternalVisible := 'False'} : Bool := FALSE;   // I67.6
      "I67.7" { ExternalVisible := 'False'} : Bool := FALSE;   // I67.7
      "I68.0" { ExternalVisible := 'False'} : Bool := FALSE;   // I68.0
      "I68.1" { ExternalVisible := 'False'} : Bool := FALSE;   // I68.1
      "I68.2" { ExternalVisible := 'False'} : Bool := FALSE;   // I68.2
      "I68.3" { ExternalVisible := 'False'} : Bool := FALSE;   // I68.3
      "I68.4" { ExternalVisible := 'False'} : Bool := FALSE;   // I68.4
      "I68.5" { ExternalVisible := 'False'} : Bool := FALSE;   // I68.5
      "I68.6" { ExternalVisible := 'False'} : Bool := FALSE;   // I68.6
      "I68.7" { ExternalVisible := 'False'} : Bool := FALSE;   // I68.7
      "I69.0" { ExternalVisible := 'False'} : Bool := FALSE;   // I69.0
      "I69.1" { ExternalVisible := 'False'} : Bool := FALSE;   // I69.1
      "I69.2" { ExternalVisible := 'False'} : Bool := FALSE;   // I69.2
      "I69.3" { ExternalVisible := 'False'} : Bool := FALSE;   // I69.3
      "I69.4" { ExternalVisible := 'False'} : Bool := FALSE;   // I69.4
      "I69.5" { ExternalVisible := 'False'} : Bool := FALSE;   // I69.5
      "I69.6" { ExternalVisible := 'False'} : Bool := FALSE;   // I69.6
      "I69.7" { ExternalVisible := 'False'} : Bool := FALSE;   // I69.7
      "I70.0" { ExternalVisible := 'False'} : Bool := FALSE;   // I70.0
      "I70.1" { ExternalVisible := 'False'} : Bool := FALSE;   // I70.1
      "I70.2" { ExternalVisible := 'False'} : Bool := FALSE;   // I70.2
      "I70.3" { ExternalVisible := 'False'} : Bool := FALSE;   // I70.3
      "I70.4" { ExternalVisible := 'False'} : Bool := FALSE;   // I70.4
      "I70.5" { ExternalVisible := 'False'} : Bool := FALSE;   // I70.5
      "I70.6" { ExternalVisible := 'False'} : Bool := FALSE;   // I70.6
      "I70.7" { ExternalVisible := 'False'} : Bool := FALSE;   // I70.7
      "I71.0" { ExternalVisible := 'False'} : Bool := FALSE;   // I71.0
      "I71.1" { ExternalVisible := 'False'} : Bool := FALSE;   // I71.1
      "I71.2" { ExternalVisible := 'False'} : Bool := FALSE;   // I71.2
      "I71.3" { ExternalVisible := 'False'} : Bool := FALSE;   // I71.3
      "I71.4" { ExternalVisible := 'False'} : Bool := FALSE;   // I71.4
      "I71.5" { ExternalVisible := 'False'} : Bool := FALSE;   // I71.5
      "I71.6" { ExternalVisible := 'False'} : Bool := FALSE;   // I71.6
      "I71.7" { ExternalVisible := 'False'} : Bool := FALSE;   // I71.7
      "I72.0" { ExternalVisible := 'False'} : Bool := FALSE;   // I72.0
      "I72.1" { ExternalVisible := 'False'} : Bool := FALSE;   // I72.1
      "I72.2" { ExternalVisible := 'False'} : Bool := FALSE;   // I72.2
      "I72.3" { ExternalVisible := 'False'} : Bool := FALSE;   // I72.3
      "I72.4" { ExternalVisible := 'False'} : Bool := FALSE;   // I72.4
      "I72.5" { ExternalVisible := 'False'} : Bool := FALSE;   // I72.5
      "I72.6" { ExternalVisible := 'False'} : Bool := FALSE;   // I72.6
      "I72.7" { ExternalVisible := 'False'} : Bool := FALSE;   // I72.7
      "I73.0" { ExternalVisible := 'False'} : Bool := FALSE;   // I73.0
      "I73.1" { ExternalVisible := 'False'} : Bool := FALSE;   // I73.1
      "I73.2" { ExternalVisible := 'False'} : Bool := FALSE;   // I73.2
      "I73.3" { ExternalVisible := 'False'} : Bool := FALSE;   // I73.3
      "I73.4" { ExternalVisible := 'False'} : Bool := FALSE;   // I73.4
      "I73.5" { ExternalVisible := 'False'} : Bool := FALSE;   // I73.5
      "I73.6" { ExternalVisible := 'False'} : Bool := FALSE;   // I73.6
      "I73.7" { ExternalVisible := 'False'} : Bool := FALSE;   // I73.7
      "I74.0" { ExternalVisible := 'False'} : Bool := FALSE;   // I74.0
      "I74.1" { ExternalVisible := 'False'} : Bool := FALSE;   // I74.1
      "I74.2" { ExternalVisible := 'False'} : Bool := FALSE;   // I74.2
      "I74.3" { ExternalVisible := 'False'} : Bool := FALSE;   // I74.3
      "I74.4" { ExternalVisible := 'False'} : Bool := FALSE;   // I74.4
      "I74.5" { ExternalVisible := 'False'} : Bool := FALSE;   // I74.5
      "I74.6" { ExternalVisible := 'False'} : Bool := FALSE;   // I74.6
      "I74.7" { ExternalVisible := 'False'} : Bool := FALSE;   // I74.7
      "I75.0" { ExternalVisible := 'False'} : Bool := FALSE;   // I75.0
      "I75.1" { ExternalVisible := 'False'} : Bool := FALSE;   // I75.1
      "I75.2" { ExternalVisible := 'False'} : Bool := FALSE;   // I75.2
      "I75.3" { ExternalVisible := 'False'} : Bool := FALSE;   // I75.3
      "I75.4" { ExternalVisible := 'False'} : Bool := FALSE;   // I75.4
      "I75.5" { ExternalVisible := 'False'} : Bool := FALSE;   // I75.5
      "I75.6" { ExternalVisible := 'False'} : Bool := FALSE;   // I75.6
      "I75.7" { ExternalVisible := 'False'} : Bool := FALSE;   // I75.7
      "I76.0" { ExternalVisible := 'False'} : Bool := FALSE;   // I76.0
      "I76.1" { ExternalVisible := 'False'} : Bool := FALSE;   // I76.1
      "I76.2" { ExternalVisible := 'False'} : Bool := FALSE;   // I76.2
      "I76.3" { ExternalVisible := 'False'} : Bool := FALSE;   // I76.3
      "I76.4" { ExternalVisible := 'False'} : Bool := FALSE;   // I76.4
      "I76.5" { ExternalVisible := 'False'} : Bool := FALSE;   // I76.5
      "I76.6" { ExternalVisible := 'False'} : Bool := FALSE;   // I76.6
      "I76.7" { ExternalVisible := 'False'} : Bool := FALSE;   // I76.7
      "I77.0" { ExternalVisible := 'False'} : Bool := FALSE;   // I77.0
      "I77.1" { ExternalVisible := 'False'} : Bool := FALSE;   // I77.1
      "I77.2" { ExternalVisible := 'False'} : Bool := FALSE;   // I77.2
      "I77.3" { ExternalVisible := 'False'} : Bool := FALSE;   // I77.3
      "I77.4" { ExternalVisible := 'False'} : Bool := FALSE;   // I77.4
      "I77.5" { ExternalVisible := 'False'} : Bool := FALSE;   // I77.5
      "I77.6" { ExternalVisible := 'False'} : Bool := FALSE;   // I77.6
      "I77.7" { ExternalVisible := 'False'} : Bool := FALSE;   // I77.7
      "I78.0" { ExternalVisible := 'False'} : Bool := FALSE;   // I78.0
      "I78.1" { ExternalVisible := 'False'} : Bool := FALSE;   // I78.1
      "I78.2" { ExternalVisible := 'False'} : Bool := FALSE;   // I78.2
      "I78.3" { ExternalVisible := 'False'} : Bool := FALSE;   // I78.3
      "I78.4" { ExternalVisible := 'False'} : Bool := FALSE;   // I78.4
      "I78.5" { ExternalVisible := 'False'} : Bool := FALSE;   // I78.5
      "I78.6" { ExternalVisible := 'False'} : Bool := FALSE;   // I78.6
      "I78.7" { ExternalVisible := 'False'} : Bool := FALSE;   // I78.7
      "I79.0" { ExternalVisible := 'False'} : Bool := FALSE;   // I79.0
      "I79.1" { ExternalVisible := 'False'} : Bool := FALSE;   // I79.1
      "I79.2" { ExternalVisible := 'False'} : Bool := FALSE;   // I79.2
      "I79.3" { ExternalVisible := 'False'} : Bool := FALSE;   // I79.3
      "I79.4" { ExternalVisible := 'False'} : Bool := FALSE;   // I79.4
      "I79.5" { ExternalVisible := 'False'} : Bool := FALSE;   // I79.5
      "I79.6" { ExternalVisible := 'False'} : Bool := FALSE;   // I79.6
      "I79.7" { ExternalVisible := 'False'} : Bool := FALSE;   // I79.7
      "I80.0" { ExternalVisible := 'False'} : Bool := FALSE;   // I80.0
      "I80.1" { ExternalVisible := 'False'} : Bool := FALSE;   // I80.1
      "I80.2" { ExternalVisible := 'False'} : Bool := FALSE;   // I80.2
      "I80.3" { ExternalVisible := 'False'} : Bool := FALSE;   // I80.3
      "I80.4" { ExternalVisible := 'False'} : Bool := FALSE;   // I80.4
      "I80.5" { ExternalVisible := 'False'} : Bool := FALSE;   // I80.5
      "I80.6" { ExternalVisible := 'False'} : Bool := FALSE;   // I80.6
      "I80.7" { ExternalVisible := 'False'} : Bool := FALSE;   // I80.7
      "I81.0" { ExternalVisible := 'False'} : Bool := FALSE;   // I81.0
      "I81.1" { ExternalVisible := 'False'} : Bool := FALSE;   // I81.1
      "I81.2" { ExternalVisible := 'False'} : Bool := FALSE;   // I81.2
      "I81.3" { ExternalVisible := 'False'} : Bool := FALSE;   // I81.3
      "I81.4" { ExternalVisible := 'False'} : Bool := FALSE;   // I81.4
      "I81.5" { ExternalVisible := 'False'} : Bool := FALSE;   // I81.5
      "I81.6" { ExternalVisible := 'False'} : Bool := FALSE;   // I81.6
      "I81.7" { ExternalVisible := 'False'} : Bool := FALSE;   // I81.7
      "I82.0" { ExternalVisible := 'False'} : Bool := FALSE;   // I82.0
      "I82.1" { ExternalVisible := 'False'} : Bool := FALSE;   // I82.1
      "I82.2" { ExternalVisible := 'False'} : Bool := FALSE;   // I82.2
      "I82.3" { ExternalVisible := 'False'} : Bool := FALSE;   // I82.3
      "I82.4" { ExternalVisible := 'False'} : Bool := FALSE;   // I82.4
      "I82.5" { ExternalVisible := 'False'} : Bool := FALSE;   // I82.5
      "I82.6" { ExternalVisible := 'False'} : Bool := FALSE;   // I82.6
      "I82.7" { ExternalVisible := 'False'} : Bool := FALSE;   // I82.7
      "I83.0" { ExternalVisible := 'False'} : Bool := FALSE;   // I83.0
      "I83.1" { ExternalVisible := 'False'} : Bool := FALSE;   // I83.1
      "I83.2" { ExternalVisible := 'False'} : Bool := FALSE;   // I83.2
      "I83.3" { ExternalVisible := 'False'} : Bool := FALSE;   // I83.3
      "I83.4" { ExternalVisible := 'False'} : Bool := FALSE;   // I83.4
      "I83.5" { ExternalVisible := 'False'} : Bool := FALSE;   // I83.5
      "I83.6" { ExternalVisible := 'False'} : Bool := FALSE;   // I83.6
      "I83.7" { ExternalVisible := 'False'} : Bool := FALSE;   // I83.7
      "I84.0" { ExternalVisible := 'False'} : Bool := FALSE;   // I84.0
      "I84.1" { ExternalVisible := 'False'} : Bool := FALSE;   // I84.1
      "I84.2" { ExternalVisible := 'False'} : Bool := FALSE;   // I84.2
      "I84.3" { ExternalVisible := 'False'} : Bool := FALSE;   // I84.3
      "I84.4" { ExternalVisible := 'False'} : Bool := FALSE;   // I84.4
      "I84.5" { ExternalVisible := 'False'} : Bool := FALSE;   // I84.5
      "I84.6" { ExternalVisible := 'False'} : Bool := FALSE;   // I84.6
      "I84.7" { ExternalVisible := 'False'} : Bool := FALSE;   // I84.7
      "I85.0" { ExternalVisible := 'False'} : Bool := FALSE;   // I85.0
      "I85.1" { ExternalVisible := 'False'} : Bool := FALSE;   // I85.1
      "I85.2" { ExternalVisible := 'False'} : Bool := FALSE;   // I85.2
      "I85.3" { ExternalVisible := 'False'} : Bool := FALSE;   // I85.3
      "I85.4" { ExternalVisible := 'False'} : Bool := FALSE;   // I85.4
      "I85.5" { ExternalVisible := 'False'} : Bool := FALSE;   // I85.5
      "I85.6" { ExternalVisible := 'False'} : Bool := FALSE;   // I85.6
      "I85.7" { ExternalVisible := 'False'} : Bool := FALSE;   // I85.7
      "I86.0" { ExternalVisible := 'False'} : Bool := FALSE;   // I86.0
      "I86.1" { ExternalVisible := 'False'} : Bool := FALSE;   // I86.1
      "I86.2" { ExternalVisible := 'False'} : Bool := FALSE;   // I86.2
      "I86.3" { ExternalVisible := 'False'} : Bool := FALSE;   // I86.3
      "I86.4" { ExternalVisible := 'False'} : Bool := FALSE;   // I86.4
      "I86.5" { ExternalVisible := 'False'} : Bool := FALSE;   // I86.5
      "I86.6" { ExternalVisible := 'False'} : Bool := FALSE;   // I86.6
      "I86.7" { ExternalVisible := 'False'} : Bool := FALSE;   // I86.7
      "I87.0" { ExternalVisible := 'False'} : Bool := FALSE;   // I87.0
      "I87.1" { ExternalVisible := 'False'} : Bool := FALSE;   // I87.1
      "I87.2" { ExternalVisible := 'False'} : Bool := FALSE;   // I87.2
      "I87.3" { ExternalVisible := 'False'} : Bool := FALSE;   // I87.3
      "I87.4" { ExternalVisible := 'False'} : Bool := FALSE;   // I87.4
      "I87.5" { ExternalVisible := 'False'} : Bool := FALSE;   // I87.5
      "I87.6" { ExternalVisible := 'False'} : Bool := FALSE;   // I87.6
      "I87.7" { ExternalVisible := 'False'} : Bool := FALSE;   // I87.7
      "I88.0" { ExternalVisible := 'False'} : Bool := FALSE;   // I88.0
      "I88.1" { ExternalVisible := 'False'} : Bool := FALSE;   // I88.1
      "I88.2" { ExternalVisible := 'False'} : Bool := FALSE;   // I88.2
      "I88.3" { ExternalVisible := 'False'} : Bool := FALSE;   // I88.3
      "I88.4" { ExternalVisible := 'False'} : Bool := FALSE;   // I88.4
      "I88.5" { ExternalVisible := 'False'} : Bool := FALSE;   // I88.5
      "I88.6" { ExternalVisible := 'False'} : Bool := FALSE;   // I88.6
      "I88.7" { ExternalVisible := 'False'} : Bool := FALSE;   // I88.7
      "I89.0" { ExternalVisible := 'False'} : Bool := FALSE;   // I89.0
      "I89.1" { ExternalVisible := 'False'} : Bool := FALSE;   // I89.1
      "I89.2" { ExternalVisible := 'False'} : Bool := FALSE;   // I89.2
      "I89.3" { ExternalVisible := 'False'} : Bool := FALSE;   // I89.3
      "I89.4" { ExternalVisible := 'False'} : Bool := FALSE;   // I89.4
      "I89.5" { ExternalVisible := 'False'} : Bool := FALSE;   // I89.5
      "I89.6" { ExternalVisible := 'False'} : Bool := FALSE;   // I89.6
      "I89.7" { ExternalVisible := 'False'} : Bool := FALSE;   // I89.7
      "I90.0" { ExternalVisible := 'False'} : Bool := FALSE;   // I90.0
      "I90.1" { ExternalVisible := 'False'} : Bool := FALSE;   // I90.1
      "I90.2" { ExternalVisible := 'False'} : Bool := FALSE;   // I90.2
      "I90.3" { ExternalVisible := 'False'} : Bool := FALSE;   // I90.3
      "I90.4" { ExternalVisible := 'False'} : Bool := FALSE;   // I90.4
      "I90.5" { ExternalVisible := 'False'} : Bool := FALSE;   // I90.5
      "I90.6" { ExternalVisible := 'False'} : Bool := FALSE;   // I90.6
      "I90.7" { ExternalVisible := 'False'} : Bool := FALSE;   // I90.7
      "I91.0" { ExternalVisible := 'False'} : Bool := FALSE;   // I91.0
      "I91.1" { ExternalVisible := 'False'} : Bool := FALSE;   // I91.1
      "I91.2" { ExternalVisible := 'False'} : Bool := FALSE;   // I91.2
      "I91.3" { ExternalVisible := 'False'} : Bool := FALSE;   // I91.3
      "I91.4" { ExternalVisible := 'False'} : Bool := FALSE;   // I91.4
      "I91.5" { ExternalVisible := 'False'} : Bool := FALSE;   // I91.5
      "I91.6" { ExternalVisible := 'False'} : Bool := FALSE;   // I91.6
      "I91.7" { ExternalVisible := 'False'} : Bool := FALSE;   // I91.7
      "I92.0" { ExternalVisible := 'False'} : Bool := FALSE;   // I92.0
      "I92.1" { ExternalVisible := 'False'} : Bool := FALSE;   // I92.1
      "I92.2" { ExternalVisible := 'False'} : Bool := FALSE;   // I92.2
      "I92.3" { ExternalVisible := 'False'} : Bool := FALSE;   // I92.3
      "I92.4" { ExternalVisible := 'False'} : Bool := FALSE;   // I92.4
      "I92.5" { ExternalVisible := 'False'} : Bool := FALSE;   // I92.5
      "I92.6" { ExternalVisible := 'False'} : Bool := FALSE;   // I92.6
      "I92.7" { ExternalVisible := 'False'} : Bool := FALSE;   // I92.7
      "I93.0" { ExternalVisible := 'False'} : Bool := FALSE;   // I93.0
      "I93.1" { ExternalVisible := 'False'} : Bool := FALSE;   // I93.1
      "I93.2" { ExternalVisible := 'False'} : Bool := FALSE;   // I93.2
      "I93.3" { ExternalVisible := 'False'} : Bool := FALSE;   // I93.3
      "I93.4" { ExternalVisible := 'False'} : Bool := FALSE;   // I93.4
      "I93.5" { ExternalVisible := 'False'} : Bool := FALSE;   // I93.5
      "I93.6" { ExternalVisible := 'False'} : Bool := FALSE;   // I93.6
      "I93.7" { ExternalVisible := 'False'} : Bool := FALSE;   // I93.7
      "I94.0" { ExternalVisible := 'False'} : Bool := FALSE;   // I94.0
      "I94.1" { ExternalVisible := 'False'} : Bool := FALSE;   // I94.1
      "I94.2" { ExternalVisible := 'False'} : Bool := FALSE;   // I94.2
      "I94.3" { ExternalVisible := 'False'} : Bool := FALSE;   // I94.3
      "I94.4" { ExternalVisible := 'False'} : Bool := FALSE;   // I94.4
      "I94.5" { ExternalVisible := 'False'} : Bool := FALSE;   // I94.5
      "I94.6" { ExternalVisible := 'False'} : Bool := FALSE;   // I94.6
      "I94.7" { ExternalVisible := 'False'} : Bool := FALSE;   // I94.7
      "I95.0" { ExternalVisible := 'False'} : Bool := FALSE;   // I95.0
      "I95.1" { ExternalVisible := 'False'} : Bool := FALSE;   // I95.1
      "I95.2" { ExternalVisible := 'False'} : Bool := FALSE;   // I95.2
      "I95.3" { ExternalVisible := 'False'} : Bool := FALSE;   // I95.3
      "I95.4" { ExternalVisible := 'False'} : Bool := FALSE;   // I95.4
      "I95.5" { ExternalVisible := 'False'} : Bool := FALSE;   // I95.5
      "I95.6" { ExternalVisible := 'False'} : Bool := FALSE;   // I95.6
      "I95.7" { ExternalVisible := 'False'} : Bool := FALSE;   // I95.7
      "I96.0" { ExternalVisible := 'False'} : Bool := FALSE;   // I96.0
      "I96.1" { ExternalVisible := 'False'} : Bool := FALSE;   // I96.1
      "I96.2" { ExternalVisible := 'False'} : Bool := FALSE;   // I96.2
      "I96.3" { ExternalVisible := 'False'} : Bool := FALSE;   // I96.3
      "I96.4" { ExternalVisible := 'False'} : Bool := FALSE;   // I96.4
      "I96.5" { ExternalVisible := 'False'} : Bool := FALSE;   // I96.5
      "I96.6" { ExternalVisible := 'False'} : Bool := FALSE;   // I96.6
      "I96.7" { ExternalVisible := 'False'} : Bool := FALSE;   // I96.7
      "I97.0" { ExternalVisible := 'False'} : Bool := FALSE;   // I97.0
      "I97.1" { ExternalVisible := 'False'} : Bool := FALSE;   // I97.1
      "I97.2" { ExternalVisible := 'False'} : Bool := FALSE;   // I97.2
      "I97.3" { ExternalVisible := 'False'} : Bool := FALSE;   // I97.3
      "I97.4" { ExternalVisible := 'False'} : Bool := FALSE;   // I97.4
      "I97.5" { ExternalVisible := 'False'} : Bool := FALSE;   // I97.5
      "I97.6" { ExternalVisible := 'False'} : Bool := FALSE;   // I97.6
      "I97.7" { ExternalVisible := 'False'} : Bool := FALSE;   // I97.7
      "I98.0" { ExternalVisible := 'False'} : Bool := FALSE;   // I98.0
      "I98.1" { ExternalVisible := 'False'} : Bool := FALSE;   // I98.1
      "I98.2" { ExternalVisible := 'False'} : Bool := FALSE;   // I98.2
      "I98.3" { ExternalVisible := 'False'} : Bool := FALSE;   // I98.3
      "I98.4" { ExternalVisible := 'False'} : Bool := FALSE;   // I98.4
      "I98.5" { ExternalVisible := 'False'} : Bool := FALSE;   // I98.5
      "I98.6" { ExternalVisible := 'False'} : Bool := FALSE;   // I98.6
      "I98.7" { ExternalVisible := 'False'} : Bool := FALSE;   // I98.7
      "I99.0" { ExternalVisible := 'False'} : Bool := FALSE;   // I99.0
      "I99.1" { ExternalVisible := 'False'} : Bool := FALSE;   // I99.1
      "I99.2" { ExternalVisible := 'False'} : Bool := FALSE;   // I99.2
      "I99.3" { ExternalVisible := 'False'} : Bool := FALSE;   // I99.3
      "I99.4" { ExternalVisible := 'False'} : Bool := FALSE;   // I99.4
      "I99.5" { ExternalVisible := 'False'} : Bool := FALSE;   // I99.5
      "I99.6" { ExternalVisible := 'False'} : Bool := FALSE;   // I99.6
      "I99.7" { ExternalVisible := 'False'} : Bool := FALSE;   // I99.7
      "I100.0" { ExternalVisible := 'False'} : Bool := FALSE;   // I100.0
      "I100.1" { ExternalVisible := 'False'} : Bool := FALSE;   // I100.1
      "I100.2" { ExternalVisible := 'False'} : Bool := FALSE;   // I100.2
      "I100.3" { ExternalVisible := 'False'} : Bool := FALSE;   // I100.3
      "I100.4" { ExternalVisible := 'False'} : Bool := FALSE;   // I100.4
      "I100.5" { ExternalVisible := 'False'} : Bool := FALSE;   // I100.5
      "I100.6" { ExternalVisible := 'False'} : Bool := FALSE;   // I100.6
      "I100.7" { ExternalVisible := 'False'} : Bool := FALSE;   // I100.7
      "I101.0" { ExternalVisible := 'False'} : Bool := FALSE;   // I101.0
      "I101.1" { ExternalVisible := 'False'} : Bool := FALSE;   // I101.1
      "I101.2" { ExternalVisible := 'False'} : Bool := FALSE;   // I101.2
      "I101.3" { ExternalVisible := 'False'} : Bool := FALSE;   // I101.3
      "I101.4" { ExternalVisible := 'False'} : Bool := FALSE;   // I101.4
      "I101.5" { ExternalVisible := 'False'} : Bool := FALSE;   // I101.5
      "I101.6" { ExternalVisible := 'False'} : Bool := FALSE;   // I101.6
      "I101.7" { ExternalVisible := 'False'} : Bool := FALSE;   // I101.7
      "I102.0" { ExternalVisible := 'False'} : Bool := FALSE;   // I102.0
      "I102.1" { ExternalVisible := 'False'} : Bool := FALSE;   // I102.1
      "I102.2" { ExternalVisible := 'False'} : Bool := FALSE;   // I102.2
      "I102.3" { ExternalVisible := 'False'} : Bool := FALSE;   // I102.3
      "I102.4" { ExternalVisible := 'False'} : Bool := FALSE;   // I102.4
      "I102.5" { ExternalVisible := 'False'} : Bool := FALSE;   // I102.5
      "I102.6" { ExternalVisible := 'False'} : Bool := FALSE;   // I102.6
      "I102.7" { ExternalVisible := 'False'} : Bool := FALSE;   // I102.7
      "I103.0" { ExternalVisible := 'False'} : Bool := FALSE;   // I103.0
      "I103.1" { ExternalVisible := 'False'} : Bool := FALSE;   // I103.1
      "I103.2" { ExternalVisible := 'False'} : Bool := FALSE;   // I103.2
      "I103.3" { ExternalVisible := 'False'} : Bool := FALSE;   // I103.3
      "I103.4" { ExternalVisible := 'False'} : Bool := FALSE;   // I103.4
      "I103.5" { ExternalVisible := 'False'} : Bool := FALSE;   // I103.5
      "I103.6" { ExternalVisible := 'False'} : Bool := FALSE;   // I103.6
      "I103.7" { ExternalVisible := 'False'} : Bool := FALSE;   // I103.7
      "I104.0" { ExternalVisible := 'False'} : Bool := FALSE;   // I104.0
      "I104.1" { ExternalVisible := 'False'} : Bool := FALSE;   // I104.1
      "I104.2" { ExternalVisible := 'False'} : Bool := FALSE;   // I104.2
      "I104.3" { ExternalVisible := 'False'} : Bool := FALSE;   // I104.3
      "I104.4" { ExternalVisible := 'False'} : Bool := FALSE;   // I104.4
      "I104.5" { ExternalVisible := 'False'} : Bool := FALSE;   // I104.5
      "I104.6" { ExternalVisible := 'False'} : Bool := FALSE;   // I104.6
      "I104.7" { ExternalVisible := 'False'} : Bool := FALSE;   // I104.7
      "I105.0" { ExternalVisible := 'False'} : Bool := FALSE;   // I105.0
      "I105.1" { ExternalVisible := 'False'} : Bool := FALSE;   // I105.1
      "I105.2" { ExternalVisible := 'False'} : Bool := FALSE;   // I105.2
      "I105.3" { ExternalVisible := 'False'} : Bool := FALSE;   // I105.3
      "I105.4" { ExternalVisible := 'False'} : Bool := FALSE;   // I105.4
      "I105.5" { ExternalVisible := 'False'} : Bool := FALSE;   // I105.5
      "I105.6" { ExternalVisible := 'False'} : Bool := FALSE;   // I105.6
      "I105.7" { ExternalVisible := 'False'} : Bool := FALSE;   // I105.7
      "I106.0" { ExternalVisible := 'False'} : Bool := FALSE;   // I106.0
      "I106.1" { ExternalVisible := 'False'} : Bool := FALSE;   // I106.1
      "I106.2" { ExternalVisible := 'False'} : Bool := FALSE;   // I106.2
      "I106.3" { ExternalVisible := 'False'} : Bool := FALSE;   // I106.3
      "I106.4" { ExternalVisible := 'False'} : Bool := FALSE;   // I106.4
      "I106.5" { ExternalVisible := 'False'} : Bool := FALSE;   // I106.5
      "I106.6" { ExternalVisible := 'False'} : Bool := FALSE;   // I106.6
      "I106.7" { ExternalVisible := 'False'} : Bool := FALSE;   // I106.7
      "I107.0" { ExternalVisible := 'False'} : Bool := FALSE;   // I107.0
      "I107.1" { ExternalVisible := 'False'} : Bool := FALSE;   // I107.1
      "I107.2" { ExternalVisible := 'False'} : Bool := FALSE;   // I107.2
      "I107.3" { ExternalVisible := 'False'} : Bool := FALSE;   // I107.3
      "I107.4" { ExternalVisible := 'False'} : Bool := FALSE;   // I107.4
      "I107.5" { ExternalVisible := 'False'} : Bool := FALSE;   // I107.5
      "I107.6" { ExternalVisible := 'False'} : Bool := FALSE;   // I107.6
      "I107.7" { ExternalVisible := 'False'} : Bool := FALSE;   // I107.7
      "I108.0" { ExternalVisible := 'False'} : Bool := FALSE;   // I108.0
      "I108.1" { ExternalVisible := 'False'} : Bool := FALSE;   // I108.1
      "I108.2" { ExternalVisible := 'False'} : Bool := FALSE;   // I108.2
      "I108.3" { ExternalVisible := 'False'} : Bool := FALSE;   // I108.3
      "I108.4" { ExternalVisible := 'False'} : Bool := FALSE;   // I108.4
      "I108.5" { ExternalVisible := 'False'} : Bool := FALSE;   // I108.5
      "I108.6" { ExternalVisible := 'False'} : Bool := FALSE;   // I108.6
      "I108.7" { ExternalVisible := 'False'} : Bool := FALSE;   // I108.7
      "I109.0" { ExternalVisible := 'False'} : Bool := FALSE;   // I109.0
      "I109.1" { ExternalVisible := 'False'} : Bool := FALSE;   // I109.1
      "I109.2" { ExternalVisible := 'False'} : Bool := FALSE;   // I109.2
      "I109.3" { ExternalVisible := 'False'} : Bool := FALSE;   // I109.3
      "I109.4" { ExternalVisible := 'False'} : Bool := FALSE;   // I109.4
      "I109.5" { ExternalVisible := 'False'} : Bool := FALSE;   // I109.5
      "I109.6" { ExternalVisible := 'False'} : Bool := FALSE;   // I109.6
      "I109.7" { ExternalVisible := 'False'} : Bool := FALSE;   // I109.7
      "I110.0" { ExternalVisible := 'False'} : Bool := FALSE;   // I110.0
      "I110.1" { ExternalVisible := 'False'} : Bool := FALSE;   // I110.1
      "I110.2" { ExternalVisible := 'False'} : Bool := FALSE;   // I110.2
      "I110.3" { ExternalVisible := 'False'} : Bool := FALSE;   // I110.3
      "I110.4" { ExternalVisible := 'False'} : Bool := FALSE;   // I110.4
      "I110.5" { ExternalVisible := 'False'} : Bool := FALSE;   // I110.5
      "I110.6" { ExternalVisible := 'False'} : Bool := FALSE;   // I110.6
      "I110.7" { ExternalVisible := 'False'} : Bool := FALSE;   // I110.7
      "I111.0" { ExternalVisible := 'False'} : Bool := FALSE;   // I111.0
      "I111.1" { ExternalVisible := 'False'} : Bool := FALSE;   // I111.1
      "I111.2" { ExternalVisible := 'False'} : Bool := FALSE;   // I111.2
      "I111.3" { ExternalVisible := 'False'} : Bool := FALSE;   // I111.3
      "I111.4" { ExternalVisible := 'False'} : Bool := FALSE;   // I111.4
      "I111.5" { ExternalVisible := 'False'} : Bool := FALSE;   // I111.5
      "I111.6" { ExternalVisible := 'False'} : Bool := FALSE;   // I111.6
      "I111.7" { ExternalVisible := 'False'} : Bool := FALSE;   // I111.7
      "I112.0" { ExternalVisible := 'False'} : Bool := FALSE;   // I112.0
      "I112.1" { ExternalVisible := 'False'} : Bool := FALSE;   // I112.1
      "I112.2" { ExternalVisible := 'False'} : Bool := FALSE;   // I112.2
      "I112.3" { ExternalVisible := 'False'} : Bool := FALSE;   // I112.3
      "I112.4" { ExternalVisible := 'False'} : Bool := FALSE;   // I112.4
      "I112.5" { ExternalVisible := 'False'} : Bool := FALSE;   // I112.5
      "I112.6" { ExternalVisible := 'False'} : Bool := FALSE;   // I112.6
      "I112.7" { ExternalVisible := 'False'} : Bool := FALSE;   // I112.7
      "I113.0" { ExternalVisible := 'False'} : Bool := FALSE;   // I113.0
      "I113.1" { ExternalVisible := 'False'} : Bool := FALSE;   // I113.1
      "I113.2" { ExternalVisible := 'False'} : Bool := FALSE;   // I113.2
      "I113.3" { ExternalVisible := 'False'} : Bool := FALSE;   // I113.3
      "I113.4" { ExternalVisible := 'False'} : Bool := FALSE;   // I113.4
      "I113.5" { ExternalVisible := 'False'} : Bool := FALSE;   // I113.5
      "I113.6" { ExternalVisible := 'False'} : Bool := FALSE;   // I113.6
      "I113.7" { ExternalVisible := 'False'} : Bool := FALSE;   // I113.7
      "I114.0" { ExternalVisible := 'False'} : Bool := FALSE;   // I114.0
      "I114.1" { ExternalVisible := 'False'} : Bool := FALSE;   // I114.1
      "I114.2" { ExternalVisible := 'False'} : Bool := FALSE;   // I114.2
      "I114.3" { ExternalVisible := 'False'} : Bool := FALSE;   // I114.3
      "I114.4" { ExternalVisible := 'False'} : Bool := FALSE;   // I114.4
      "I114.5" { ExternalVisible := 'False'} : Bool := FALSE;   // I114.5
      "I114.6" { ExternalVisible := 'False'} : Bool := FALSE;   // I114.6
      "I114.7" { ExternalVisible := 'False'} : Bool := FALSE;   // I114.7
      "I115.0" { ExternalVisible := 'False'} : Bool := FALSE;   // I115.0
      "I115.1" { ExternalVisible := 'False'} : Bool := FALSE;   // I115.1
      "I115.2" { ExternalVisible := 'False'} : Bool := FALSE;   // I115.2
      "I115.3" { ExternalVisible := 'False'} : Bool := FALSE;   // I115.3
      "I115.4" { ExternalVisible := 'False'} : Bool := FALSE;   // I115.4
      "I115.5" { ExternalVisible := 'False'} : Bool := FALSE;   // I115.5
      "I115.6" { ExternalVisible := 'False'} : Bool := FALSE;   // I115.6
      "I115.7" { ExternalVisible := 'False'} : Bool := FALSE;   // I115.7
      "I116.0" { ExternalVisible := 'False'} : Bool := FALSE;   // I116.0
      "I116.1" { ExternalVisible := 'False'} : Bool := FALSE;   // I116.1
      "I116.2" { ExternalVisible := 'False'} : Bool := FALSE;   // I116.2
      "I116.3" { ExternalVisible := 'False'} : Bool := FALSE;   // I116.3
      "I116.4" { ExternalVisible := 'False'} : Bool := FALSE;   // I116.4
      "I116.5" { ExternalVisible := 'False'} : Bool := FALSE;   // I116.5
      "I116.6" { ExternalVisible := 'False'} : Bool := FALSE;   // I116.6
      "I116.7" { ExternalVisible := 'False'} : Bool := FALSE;   // I116.7
      "I117.0" { ExternalVisible := 'False'} : Bool := FALSE;   // I117.0
      "I117.1" { ExternalVisible := 'False'} : Bool := FALSE;   // I117.1
      "I117.2" { ExternalVisible := 'False'} : Bool := FALSE;   // I117.2
      "I117.3" { ExternalVisible := 'False'} : Bool := FALSE;   // I117.3
      "I117.4" { ExternalVisible := 'False'} : Bool := FALSE;   // I117.4
      "I117.5" { ExternalVisible := 'False'} : Bool := FALSE;   // I117.5
      "I117.6" { ExternalVisible := 'False'} : Bool := FALSE;   // I117.6
      "I117.7" { ExternalVisible := 'False'} : Bool := FALSE;   // I117.7
      "I118.0" { ExternalVisible := 'False'} : Bool := FALSE;   // I118.0
      "I118.1" { ExternalVisible := 'False'} : Bool := FALSE;   // I118.1
      "I118.2" { ExternalVisible := 'False'} : Bool := FALSE;   // I118.2
      "I118.3" { ExternalVisible := 'False'} : Bool := FALSE;   // I118.3
      "I118.4" { ExternalVisible := 'False'} : Bool := FALSE;   // I118.4
      "I118.5" { ExternalVisible := 'False'} : Bool := FALSE;   // I118.5
      "I118.6" { ExternalVisible := 'False'} : Bool := FALSE;   // I118.6
      "I118.7" { ExternalVisible := 'False'} : Bool := FALSE;   // I118.7
      "I119.0" { ExternalVisible := 'False'} : Bool := FALSE;   // I119.0
      "I119.1" { ExternalVisible := 'False'} : Bool := FALSE;   // I119.1
      "I119.2" { ExternalVisible := 'False'} : Bool := FALSE;   // I119.2
      "I119.3" { ExternalVisible := 'False'} : Bool := FALSE;   // I119.3
      "I119.4" { ExternalVisible := 'False'} : Bool := FALSE;   // I119.4
      "I119.5" { ExternalVisible := 'False'} : Bool := FALSE;   // I119.5
      "I119.6" { ExternalVisible := 'False'} : Bool := FALSE;   // I119.6
      "I119.7" { ExternalVisible := 'False'} : Bool := FALSE;   // I119.7
      "I120.0" { ExternalVisible := 'False'} : Bool := FALSE;   // I120.0
      "I120.1" { ExternalVisible := 'False'} : Bool := FALSE;   // I120.1
      "I120.2" { ExternalVisible := 'False'} : Bool := FALSE;   // I120.2
      "I120.3" { ExternalVisible := 'False'} : Bool := FALSE;   // I120.3
      "I120.4" { ExternalVisible := 'False'} : Bool := FALSE;   // I120.4
      "I120.5" { ExternalVisible := 'False'} : Bool := FALSE;   // I120.5
      "I120.6" { ExternalVisible := 'False'} : Bool := FALSE;   // I120.6
      "I120.7" { ExternalVisible := 'False'} : Bool := FALSE;   // I120.7
      "I121.0" { ExternalVisible := 'False'} : Bool := FALSE;   // I121.0
      "I121.1" { ExternalVisible := 'False'} : Bool := FALSE;   // I121.1
      "I121.2" { ExternalVisible := 'False'} : Bool := FALSE;   // I121.2
      "I121.3" { ExternalVisible := 'False'} : Bool := FALSE;   // I121.3
      "I121.4" { ExternalVisible := 'False'} : Bool := FALSE;   // I121.4
      "I121.5" { ExternalVisible := 'False'} : Bool := FALSE;   // I121.5
      "I121.6" { ExternalVisible := 'False'} : Bool := FALSE;   // I121.6
      "I121.7" { ExternalVisible := 'False'} : Bool := FALSE;   // I121.7
      "I122.0" { ExternalVisible := 'False'} : Bool := FALSE;   // I122.0
      "I122.1" { ExternalVisible := 'False'} : Bool := FALSE;   // I122.1
      "I122.2" { ExternalVisible := 'False'} : Bool := FALSE;   // I122.2
      "I122.3" { ExternalVisible := 'False'} : Bool := FALSE;   // I122.3
      "I122.4" { ExternalVisible := 'False'} : Bool := FALSE;   // I122.4
      "I122.5" { ExternalVisible := 'False'} : Bool := FALSE;   // I122.5
      "I122.6" { ExternalVisible := 'False'} : Bool := FALSE;   // I122.6
      "I122.7" { ExternalVisible := 'False'} : Bool := FALSE;   // I122.7
      "I123.0" { ExternalVisible := 'False'} : Bool := FALSE;   // I123.0
      "I123.1" { ExternalVisible := 'False'} : Bool := FALSE;   // I123.1
      "I123.2" { ExternalVisible := 'False'} : Bool := FALSE;   // I123.2
      "I123.3" { ExternalVisible := 'False'} : Bool := FALSE;   // I123.3
      "I123.4" { ExternalVisible := 'False'} : Bool := FALSE;   // I123.4
      "I123.5" { ExternalVisible := 'False'} : Bool := FALSE;   // I123.5
      "I123.6" { ExternalVisible := 'False'} : Bool := FALSE;   // I123.6
      "I123.7" { ExternalVisible := 'False'} : Bool := FALSE;   // I123.7
      "I124.0" { ExternalVisible := 'False'} : Bool := FALSE;   // I124.0
      "I124.1" { ExternalVisible := 'False'} : Bool := FALSE;   // I124.1
      "I124.2" { ExternalVisible := 'False'} : Bool := FALSE;   // I124.2
      "I124.3" { ExternalVisible := 'False'} : Bool := FALSE;   // I124.3
      "I124.4" { ExternalVisible := 'False'} : Bool := FALSE;   // I124.4
      "I124.5" { ExternalVisible := 'False'} : Bool := FALSE;   // I124.5
      "I124.6" { ExternalVisible := 'False'} : Bool := FALSE;   // I124.6
      "I124.7" { ExternalVisible := 'False'} : Bool := FALSE;   // I124.7
      "I125.0" { ExternalVisible := 'False'} : Bool := FALSE;   // I125.0
      "I125.1" { ExternalVisible := 'False'} : Bool := FALSE;   // I125.1
      "I125.2" { ExternalVisible := 'False'} : Bool := FALSE;   // I125.2
      "I125.3" { ExternalVisible := 'False'} : Bool := FALSE;   // I125.3
      "I125.4" { ExternalVisible := 'False'} : Bool := FALSE;   // I125.4
      "I125.5" { ExternalVisible := 'False'} : Bool := FALSE;   // I125.5
      "I125.6" { ExternalVisible := 'False'} : Bool := FALSE;   // I125.6
      "I125.7" { ExternalVisible := 'False'} : Bool := FALSE;   // I125.7
      "I126.0" { ExternalVisible := 'False'} : Bool := FALSE;   // I126.0
      "I126.1" { ExternalVisible := 'False'} : Bool := FALSE;   // I126.1
      "I126.2" { ExternalVisible := 'False'} : Bool := FALSE;   // I126.2
      "I126.3" { ExternalVisible := 'False'} : Bool := FALSE;   // I126.3
      "I126.4" { ExternalVisible := 'False'} : Bool := FALSE;   // I126.4
      "I126.5" { ExternalVisible := 'False'} : Bool := FALSE;   // I126.5
      "I126.6" { ExternalVisible := 'False'} : Bool := FALSE;   // I126.6
      "I126.7" { ExternalVisible := 'False'} : Bool := FALSE;   // I126.7
      "I127.0" { ExternalVisible := 'False'} : Bool := FALSE;   // I127.0
      "I127.1" { ExternalVisible := 'False'} : Bool := FALSE;   // I127.1
      "I127.2" { ExternalVisible := 'False'} : Bool := FALSE;   // I127.2
      "I127.3" { ExternalVisible := 'False'} : Bool := FALSE;   // I127.3
      "I127.4" { ExternalVisible := 'False'} : Bool := FALSE;   // I127.4
      "I127.5" { ExternalVisible := 'False'} : Bool := FALSE;   // I127.5
      "I127.6" { ExternalVisible := 'False'} : Bool := FALSE;   // I127.6
      "I127.7" { ExternalVisible := 'False'} : Bool := FALSE;   // I127.7
      "I128.0" { ExternalVisible := 'False'} : Bool := FALSE;   // I128.0
      "I128.1" { ExternalVisible := 'False'} : Bool := FALSE;   // I128.1
      "I128.2" { ExternalVisible := 'False'} : Bool := FALSE;   // I128.2
      "I128.3" { ExternalVisible := 'False'} : Bool := FALSE;   // I128.3
      "I128.4" { ExternalVisible := 'False'} : Bool := FALSE;   // I128.4
      "I128.5" { ExternalVisible := 'False'} : Bool := FALSE;   // I128.5
      "I128.6" { ExternalVisible := 'False'} : Bool := FALSE;   // I128.6
      "I128.7" { ExternalVisible := 'False'} : Bool := FALSE;   // I128.7
      "I129.0" { ExternalVisible := 'False'} : Bool := FALSE;   // I129.0
      "I129.1" { ExternalVisible := 'False'} : Bool := FALSE;   // I129.1
      "I129.2" { ExternalVisible := 'False'} : Bool := FALSE;   // I129.2
      "I129.3" { ExternalVisible := 'False'} : Bool := FALSE;   // I129.3
      "I129.4" { ExternalVisible := 'False'} : Bool := FALSE;   // I129.4
      "I129.5" { ExternalVisible := 'False'} : Bool := FALSE;   // I129.5
      "I129.6" { ExternalVisible := 'False'} : Bool := FALSE;   // I129.6
      "I129.7" { ExternalVisible := 'False'} : Bool := FALSE;   // I129.7
      "I130.0" { ExternalVisible := 'False'} : Bool := FALSE;   // I130.0
      "I130.1" { ExternalVisible := 'False'} : Bool := FALSE;   // I130.1
      "I130.2" { ExternalVisible := 'False'} : Bool := FALSE;   // I130.2
      "I130.3" { ExternalVisible := 'False'} : Bool := FALSE;   // I130.3
      "I130.4" { ExternalVisible := 'False'} : Bool := FALSE;   // I130.4
      "I130.5" { ExternalVisible := 'False'} : Bool := FALSE;   // I130.5
      "I130.6" { ExternalVisible := 'False'} : Bool := FALSE;   // I130.6
      "I130.7" { ExternalVisible := 'False'} : Bool := FALSE;   // I130.7
      "I131.0" { ExternalVisible := 'False'} : Bool := FALSE;   // I131.0
      "I131.1" { ExternalVisible := 'False'} : Bool := FALSE;   // I131.1
      "I131.2" { ExternalVisible := 'False'} : Bool := FALSE;   // I131.2
      "I131.3" { ExternalVisible := 'False'} : Bool := FALSE;   // I131.3
      "I131.4" { ExternalVisible := 'False'} : Bool := FALSE;   // I131.4
      "I131.5" { ExternalVisible := 'False'} : Bool := FALSE;   // I131.5
      "I131.6" { ExternalVisible := 'False'} : Bool := FALSE;   // I131.6
      "I131.7" { ExternalVisible := 'False'} : Bool := FALSE;   // I131.7
      "I132.0" { ExternalVisible := 'False'} : Bool := FALSE;   // I132.0
      "I132.1" { ExternalVisible := 'False'} : Bool := FALSE;   // I132.1
      "I132.2" { ExternalVisible := 'False'} : Bool := FALSE;   // I132.2
      "I132.3" { ExternalVisible := 'False'} : Bool := FALSE;   // I132.3
      "I132.4" { ExternalVisible := 'False'} : Bool := FALSE;   // I132.4
      "I132.5" { ExternalVisible := 'False'} : Bool := FALSE;   // I132.5
      "I132.6" { ExternalVisible := 'False'} : Bool := FALSE;   // I132.6
      "I132.7" { ExternalVisible := 'False'} : Bool := FALSE;   // I132.7
      "I133.0" { ExternalVisible := 'False'} : Bool := FALSE;   // I133.0
      "I133.1" { ExternalVisible := 'False'} : Bool := FALSE;   // I133.1
      "I133.2" { ExternalVisible := 'False'} : Bool := FALSE;   // I133.2
      "I133.3" { ExternalVisible := 'False'} : Bool := FALSE;   // I133.3
      "I133.4" { ExternalVisible := 'False'} : Bool := FALSE;   // I133.4
      "I133.5" { ExternalVisible := 'False'} : Bool := FALSE;   // I133.5
      "I133.6" { ExternalVisible := 'False'} : Bool := FALSE;   // I133.6
      "I133.7" { ExternalVisible := 'False'} : Bool := FALSE;   // I133.7
      "I134.0" { ExternalVisible := 'False'} : Bool := FALSE;   // I134.0
      "I134.1" { ExternalVisible := 'False'} : Bool := FALSE;   // I134.1
      "I134.2" { ExternalVisible := 'False'} : Bool := FALSE;   // I134.2
      "I134.3" { ExternalVisible := 'False'} : Bool := FALSE;   // I134.3
      "I134.4" { ExternalVisible := 'False'} : Bool := FALSE;   // I134.4
      "I134.5" { ExternalVisible := 'False'} : Bool := FALSE;   // I134.5
      "I134.6" { ExternalVisible := 'False'} : Bool := FALSE;   // I134.6
      "I134.7" { ExternalVisible := 'False'} : Bool := FALSE;   // I134.7
      "I135.0" { ExternalVisible := 'False'} : Bool := FALSE;   // I135.0
      "I135.1" { ExternalVisible := 'False'} : Bool := FALSE;   // I135.1
      "I135.2" { ExternalVisible := 'False'} : Bool := FALSE;   // I135.2
      "I135.3" { ExternalVisible := 'False'} : Bool := FALSE;   // I135.3
      "I135.4" { ExternalVisible := 'False'} : Bool := FALSE;   // I135.4
      "I135.5" { ExternalVisible := 'False'} : Bool := FALSE;   // I135.5
      "I135.6" { ExternalVisible := 'False'} : Bool := FALSE;   // I135.6
      "I135.7" { ExternalVisible := 'False'} : Bool := FALSE;   // I135.7
      "I136.0" { ExternalVisible := 'False'} : Bool := FALSE;   // I136.0
      "I136.1" { ExternalVisible := 'False'} : Bool := FALSE;   // I136.1
      "I136.2" { ExternalVisible := 'False'} : Bool := FALSE;   // I136.2
      "I136.3" { ExternalVisible := 'False'} : Bool := FALSE;   // I136.3
      "I136.4" { ExternalVisible := 'False'} : Bool := FALSE;   // I136.4
      "I136.5" { ExternalVisible := 'False'} : Bool := FALSE;   // I136.5
      "I136.6" { ExternalVisible := 'False'} : Bool := FALSE;   // I136.6
      "I136.7" { ExternalVisible := 'False'} : Bool := FALSE;   // I136.7
      "I137.0" { ExternalVisible := 'False'} : Bool := FALSE;   // I137.0
      "I137.1" { ExternalVisible := 'False'} : Bool := FALSE;   // I137.1
      "I137.2" { ExternalVisible := 'False'} : Bool := FALSE;   // I137.2
      "I137.3" { ExternalVisible := 'False'} : Bool := FALSE;   // I137.3
      "I137.4" { ExternalVisible := 'False'} : Bool := FALSE;   // I137.4
      "I137.5" { ExternalVisible := 'False'} : Bool := FALSE;   // I137.5
      "I137.6" { ExternalVisible := 'False'} : Bool := FALSE;   // I137.6
      "I137.7" { ExternalVisible := 'False'} : Bool := FALSE;   // I137.7
      "I138.0" { ExternalVisible := 'False'} : Bool := FALSE;   // I138.0
      "I138.1" { ExternalVisible := 'False'} : Bool := FALSE;   // I138.1
      "I138.2" { ExternalVisible := 'False'} : Bool := FALSE;   // I138.2
      "I138.3" { ExternalVisible := 'False'} : Bool := FALSE;   // I138.3
      "I138.4" { ExternalVisible := 'False'} : Bool := FALSE;   // I138.4
      "I138.5" { ExternalVisible := 'False'} : Bool := FALSE;   // I138.5
      "I138.6" { ExternalVisible := 'False'} : Bool := FALSE;   // I138.6
      "I138.7" { ExternalVisible := 'False'} : Bool := FALSE;   // I138.7
      "I139.0" { ExternalVisible := 'False'} : Bool := FALSE;   // I139.0
      "I139.1" { ExternalVisible := 'False'} : Bool := FALSE;   // I139.1
      "I139.2" { ExternalVisible := 'False'} : Bool := FALSE;   // I139.2
      "I139.3" { ExternalVisible := 'False'} : Bool := FALSE;   // I139.3
      "I139.4" { ExternalVisible := 'False'} : Bool := FALSE;   // I139.4
      "I139.5" { ExternalVisible := 'False'} : Bool := FALSE;   // I139.5
      "I139.6" { ExternalVisible := 'False'} : Bool := FALSE;   // I139.6
      "I139.7" { ExternalVisible := 'False'} : Bool := FALSE;   // I139.7
      "I140.0" { ExternalVisible := 'False'} : Bool := FALSE;   // I140.0
      "I140.1" { ExternalVisible := 'False'} : Bool := FALSE;   // I140.1
      "I140.2" { ExternalVisible := 'False'} : Bool := FALSE;   // I140.2
      "I140.3" { ExternalVisible := 'False'} : Bool := FALSE;   // I140.3
      "I140.4" { ExternalVisible := 'False'} : Bool := FALSE;   // I140.4
      "I140.5" { ExternalVisible := 'False'} : Bool := FALSE;   // I140.5
      "I140.6" { ExternalVisible := 'False'} : Bool := FALSE;   // I140.6
      "I140.7" { ExternalVisible := 'False'} : Bool := FALSE;   // I140.7
      "I141.0" { ExternalVisible := 'False'} : Bool := FALSE;   // I141.0
      "I141.1" { ExternalVisible := 'False'} : Bool := FALSE;   // I141.1
      "I141.2" { ExternalVisible := 'False'} : Bool := FALSE;   // I141.2
      "I141.3" { ExternalVisible := 'False'} : Bool := FALSE;   // I141.3
      "I141.4" { ExternalVisible := 'False'} : Bool := FALSE;   // I141.4
      "I141.5" { ExternalVisible := 'False'} : Bool := FALSE;   // I141.5
      "I141.6" { ExternalVisible := 'False'} : Bool := FALSE;   // I141.6
      "I141.7" { ExternalVisible := 'False'} : Bool := FALSE;   // I141.7
      "I142.0" { ExternalVisible := 'False'} : Bool := FALSE;   // I142.0
      "I142.1" { ExternalVisible := 'False'} : Bool := FALSE;   // I142.1
      "I142.2" { ExternalVisible := 'False'} : Bool := FALSE;   // I142.2
      "I142.3" { ExternalVisible := 'False'} : Bool := FALSE;   // I142.3
      "I142.4" { ExternalVisible := 'False'} : Bool := FALSE;   // I142.4
      "I142.5" { ExternalVisible := 'False'} : Bool := FALSE;   // I142.5
      "I142.6" { ExternalVisible := 'False'} : Bool := FALSE;   // I142.6
      "I142.7" { ExternalVisible := 'False'} : Bool := FALSE;   // I142.7
      "I143.0" { ExternalVisible := 'False'} : Bool := FALSE;   // I143.0
      "I143.1" { ExternalVisible := 'False'} : Bool := FALSE;   // I143.1
      "I143.2" { ExternalVisible := 'False'} : Bool := FALSE;   // I143.2
      "I143.3" { ExternalVisible := 'False'} : Bool := FALSE;   // I143.3
      "I143.4" { ExternalVisible := 'False'} : Bool := FALSE;   // I143.4
      "I143.5" { ExternalVisible := 'False'} : Bool := FALSE;   // I143.5
      "I143.6" { ExternalVisible := 'False'} : Bool := FALSE;   // I143.6
      "I143.7" { ExternalVisible := 'False'} : Bool := FALSE;   // I143.7
      "I144.0" { ExternalVisible := 'False'} : Bool := FALSE;   // I144.0
      "I144.1" { ExternalVisible := 'False'} : Bool := FALSE;   // I144.1
      "I144.2" { ExternalVisible := 'False'} : Bool := FALSE;   // I144.2
      "I144.3" { ExternalVisible := 'False'} : Bool := FALSE;   // I144.3
      "I144.4" { ExternalVisible := 'False'} : Bool := FALSE;   // I144.4
      "I144.5" { ExternalVisible := 'False'} : Bool := FALSE;   // I144.5
      "I144.6" { ExternalVisible := 'False'} : Bool := FALSE;   // I144.6
      "I144.7" { ExternalVisible := 'False'} : Bool := FALSE;   // I144.7
      "I145.0" { ExternalVisible := 'False'} : Bool := FALSE;   // I145.0
      "I145.1" { ExternalVisible := 'False'} : Bool := FALSE;   // I145.1
      "I145.2" { ExternalVisible := 'False'} : Bool := FALSE;   // I145.2
      "I145.3" { ExternalVisible := 'False'} : Bool := FALSE;   // I145.3
      "I145.4" { ExternalVisible := 'False'} : Bool := FALSE;   // I145.4
      "I145.5" { ExternalVisible := 'False'} : Bool := FALSE;   // I145.5
      "I145.6" { ExternalVisible := 'False'} : Bool := FALSE;   // I145.6
      "I145.7" { ExternalVisible := 'False'} : Bool := FALSE;   // I145.7
      "I146.0" { ExternalVisible := 'False'} : Bool := FALSE;   // I146.0
      "I146.1" { ExternalVisible := 'False'} : Bool := FALSE;   // I146.1
      "I146.2" { ExternalVisible := 'False'} : Bool := FALSE;   // I146.2
      "I146.3" { ExternalVisible := 'False'} : Bool := FALSE;   // I146.3
      "I146.4" { ExternalVisible := 'False'} : Bool := FALSE;   // I146.4
      "I146.5" { ExternalVisible := 'False'} : Bool := FALSE;   // I146.5
      "I146.6" { ExternalVisible := 'False'} : Bool := FALSE;   // I146.6
      "I146.7" { ExternalVisible := 'False'} : Bool := FALSE;   // I146.7
      "I147.0" { ExternalVisible := 'False'} : Bool := FALSE;   // I147.0
      "I147.1" { ExternalVisible := 'False'} : Bool := FALSE;   // I147.1
      "I147.2" { ExternalVisible := 'False'} : Bool := FALSE;   // I147.2
      "I147.3" { ExternalVisible := 'False'} : Bool := FALSE;   // I147.3
      "I147.4" { ExternalVisible := 'False'} : Bool := FALSE;   // I147.4
      "I147.5" { ExternalVisible := 'False'} : Bool := FALSE;   // I147.5
      "I147.6" { ExternalVisible := 'False'} : Bool := FALSE;   // I147.6
      "I147.7" { ExternalVisible := 'False'} : Bool := FALSE;   // I147.7
      "I148.0" { ExternalVisible := 'False'} : Bool := FALSE;   // I148.0
      "I148.1" { ExternalVisible := 'False'} : Bool := FALSE;   // I148.1
      "I148.2" { ExternalVisible := 'False'} : Bool := FALSE;   // I148.2
      "I148.3" { ExternalVisible := 'False'} : Bool := FALSE;   // I148.3
      "I148.4" { ExternalVisible := 'False'} : Bool := FALSE;   // I148.4
      "I148.5" { ExternalVisible := 'False'} : Bool := FALSE;   // I148.5
      "I148.6" { ExternalVisible := 'False'} : Bool := FALSE;   // I148.6
      "I148.7" { ExternalVisible := 'False'} : Bool := FALSE;   // I148.7
      "I149.0" { ExternalVisible := 'False'} : Bool := FALSE;   // I149.0
      "I149.1" { ExternalVisible := 'False'} : Bool := FALSE;   // I149.1
      "I149.2" { ExternalVisible := 'False'} : Bool := FALSE;   // I149.2
      "I149.3" { ExternalVisible := 'False'} : Bool := FALSE;   // I149.3
      "I149.4" { ExternalVisible := 'False'} : Bool := FALSE;   // I149.4
      "I149.5" { ExternalVisible := 'False'} : Bool := FALSE;   // I149.5
      "I149.6" { ExternalVisible := 'False'} : Bool := FALSE;   // I149.6
      "I149.7" { ExternalVisible := 'False'} : Bool := FALSE;   // I149.7
      "I150.0" { ExternalVisible := 'False'} : Bool := FALSE;   // I150.0
      "I150.1" { ExternalVisible := 'False'} : Bool := FALSE;   // I150.1
      "I150.2" { ExternalVisible := 'False'} : Bool := FALSE;   // I150.2
      "I150.3" { ExternalVisible := 'False'} : Bool := FALSE;   // I150.3
      "I150.4" { ExternalVisible := 'False'} : Bool := FALSE;   // I150.4
      "I150.5" { ExternalVisible := 'False'} : Bool := FALSE;   // I150.5
      "I150.6" { ExternalVisible := 'False'} : Bool := FALSE;   // I150.6
      "I150.7" { ExternalVisible := 'False'} : Bool := FALSE;   // I150.7
      "I151.0" { ExternalVisible := 'False'} : Bool := FALSE;   // I151.0
      "I151.1" { ExternalVisible := 'False'} : Bool := FALSE;   // I151.1
      "I151.2" { ExternalVisible := 'False'} : Bool := FALSE;   // I151.2
      "I151.3" { ExternalVisible := 'False'} : Bool := FALSE;   // I151.3
      "I151.4" { ExternalVisible := 'False'} : Bool := FALSE;   // I151.4
      "I151.5" { ExternalVisible := 'False'} : Bool := FALSE;   // I151.5
      "I151.6" { ExternalVisible := 'False'} : Bool := FALSE;   // I151.6
      "I151.7" { ExternalVisible := 'False'} : Bool := FALSE;   // I151.7
      "I152.0" { ExternalVisible := 'False'} : Bool := FALSE;   // I152.0
      "I152.1" { ExternalVisible := 'False'} : Bool := FALSE;   // I152.1
      "I152.2" { ExternalVisible := 'False'} : Bool := FALSE;   // I152.2
      "I152.3" { ExternalVisible := 'False'} : Bool := FALSE;   // I152.3
      "I152.4" { ExternalVisible := 'False'} : Bool := FALSE;   // I152.4
      "I152.5" { ExternalVisible := 'False'} : Bool := FALSE;   // I152.5
      "I152.6" { ExternalVisible := 'False'} : Bool := FALSE;   // I152.6
      "I152.7" { ExternalVisible := 'False'} : Bool := FALSE;   // I152.7
      "I153.0" { ExternalVisible := 'False'} : Bool := FALSE;   // I153.0
      "I153.1" { ExternalVisible := 'False'} : Bool := FALSE;   // I153.1
      "I153.2" { ExternalVisible := 'False'} : Bool := FALSE;   // I153.2
      "I153.3" { ExternalVisible := 'False'} : Bool := FALSE;   // I153.3
      "I153.4" { ExternalVisible := 'False'} : Bool := FALSE;   // I153.4
      "I153.5" { ExternalVisible := 'False'} : Bool := FALSE;   // I153.5
      "I153.6" { ExternalVisible := 'False'} : Bool := FALSE;   // I153.6
      "I153.7" { ExternalVisible := 'False'} : Bool := FALSE;   // I153.7
      "I154.0" { ExternalVisible := 'False'} : Bool := FALSE;   // I154.0
      "I154.1" { ExternalVisible := 'False'} : Bool := FALSE;   // I154.1
      "I154.2" { ExternalVisible := 'False'} : Bool := FALSE;   // I154.2
      "I154.3" { ExternalVisible := 'False'} : Bool := FALSE;   // I154.3
      "I154.4" { ExternalVisible := 'False'} : Bool := FALSE;   // I154.4
      "I154.5" { ExternalVisible := 'False'} : Bool := FALSE;   // I154.5
      "I154.6" { ExternalVisible := 'False'} : Bool := FALSE;   // I154.6
      "I154.7" { ExternalVisible := 'False'} : Bool := FALSE;   // I154.7
      "I155.0" { ExternalVisible := 'False'} : Bool := FALSE;   // I155.0
      "I155.1" { ExternalVisible := 'False'} : Bool := FALSE;   // I155.1
      "I155.2" { ExternalVisible := 'False'} : Bool := FALSE;   // I155.2
      "I155.3" { ExternalVisible := 'False'} : Bool := FALSE;   // I155.3
      "I155.4" { ExternalVisible := 'False'} : Bool := FALSE;   // I155.4
      "I155.5" { ExternalVisible := 'False'} : Bool := FALSE;   // I155.5
      "I155.6" { ExternalVisible := 'False'} : Bool := FALSE;   // I155.6
      "I155.7" { ExternalVisible := 'False'} : Bool := FALSE;   // I155.7
      "I156.0" { ExternalVisible := 'False'} : Bool := FALSE;   // I156.0
      "I156.1" { ExternalVisible := 'False'} : Bool := FALSE;   // I156.1
      "I156.2" { ExternalVisible := 'False'} : Bool := FALSE;   // I156.2
      "I156.3" { ExternalVisible := 'False'} : Bool := FALSE;   // I156.3
      "I156.4" { ExternalVisible := 'False'} : Bool := FALSE;   // I156.4
      "I156.5" { ExternalVisible := 'False'} : Bool := FALSE;   // I156.5
      "I156.6" { ExternalVisible := 'False'} : Bool := FALSE;   // I156.6
      "I156.7" { ExternalVisible := 'False'} : Bool := FALSE;   // I156.7
      "I157.0" { ExternalVisible := 'False'} : Bool := FALSE;   // I157.0
      "I157.1" { ExternalVisible := 'False'} : Bool := FALSE;   // I157.1
      "I157.2" { ExternalVisible := 'False'} : Bool := FALSE;   // I157.2
      "I157.3" { ExternalVisible := 'False'} : Bool := FALSE;   // I157.3
      "I157.4" { ExternalVisible := 'False'} : Bool := FALSE;   // I157.4
      "I157.5" { ExternalVisible := 'False'} : Bool := FALSE;   // I157.5
      "I157.6" { ExternalVisible := 'False'} : Bool := FALSE;   // I157.6
      "I157.7" { ExternalVisible := 'False'} : Bool := FALSE;   // I157.7
      "I158.0" { ExternalVisible := 'False'} : Bool := FALSE;   // I158.0
      "I158.1" { ExternalVisible := 'False'} : Bool := FALSE;   // I158.1
      "I158.2" { ExternalVisible := 'False'} : Bool := FALSE;   // I158.2
      "I158.3" { ExternalVisible := 'False'} : Bool := FALSE;   // I158.3
      "I158.4" { ExternalVisible := 'False'} : Bool := FALSE;   // I158.4
      "I158.5" { ExternalVisible := 'False'} : Bool := FALSE;   // I158.5
      "I158.6" { ExternalVisible := 'False'} : Bool := FALSE;   // I158.6
      "I158.7" { ExternalVisible := 'False'} : Bool := FALSE;   // I158.7
      "I159.0" { ExternalVisible := 'False'} : Bool := FALSE;   // I159.0
      "I159.1" { ExternalVisible := 'False'} : Bool := FALSE;   // I159.1
      "I159.2" { ExternalVisible := 'False'} : Bool := FALSE;   // I159.2
      "I159.3" { ExternalVisible := 'False'} : Bool := FALSE;   // I159.3
      "I159.4" { ExternalVisible := 'False'} : Bool := FALSE;   // I159.4
      "I159.5" { ExternalVisible := 'False'} : Bool := FALSE;   // I159.5
      "I159.6" { ExternalVisible := 'False'} : Bool := FALSE;   // I159.6
      "I159.7" { ExternalVisible := 'False'} : Bool := FALSE;   // I159.7
      "I160.0" { ExternalVisible := 'False'} : Bool := FALSE;   // I160.0
      "I160.1" { ExternalVisible := 'False'} : Bool := FALSE;   // I160.1
      "I160.2" { ExternalVisible := 'False'} : Bool := FALSE;   // I160.2
      "I160.3" { ExternalVisible := 'False'} : Bool := FALSE;   // I160.3
      "I160.4" { ExternalVisible := 'False'} : Bool := FALSE;   // I160.4
      "I160.5" { ExternalVisible := 'False'} : Bool := FALSE;   // I160.5
      "I160.6" { ExternalVisible := 'False'} : Bool := FALSE;   // I160.6
      "I160.7" { ExternalVisible := 'False'} : Bool := FALSE;   // I160.7
      "I161.0" { ExternalVisible := 'False'} : Bool := FALSE;   // I161.0
      "I161.1" { ExternalVisible := 'False'} : Bool := FALSE;   // I161.1
      "I161.2" { ExternalVisible := 'False'} : Bool := FALSE;   // I161.2
      "I161.3" { ExternalVisible := 'False'} : Bool := FALSE;   // I161.3
      "I161.4" { ExternalVisible := 'False'} : Bool := FALSE;   // I161.4
      "I161.5" { ExternalVisible := 'False'} : Bool := FALSE;   // I161.5
      "I161.6" { ExternalVisible := 'False'} : Bool := FALSE;   // I161.6
      "I161.7" { ExternalVisible := 'False'} : Bool := FALSE;   // I161.7
      "I162.0" { ExternalVisible := 'False'} : Bool := FALSE;   // I162.0
      "I162.1" { ExternalVisible := 'False'} : Bool := FALSE;   // I162.1
      "I162.2" { ExternalVisible := 'False'} : Bool := FALSE;   // I162.2
      "I162.3" { ExternalVisible := 'False'} : Bool := FALSE;   // I162.3
      "I162.4" { ExternalVisible := 'False'} : Bool := FALSE;   // I162.4
      "I162.5" { ExternalVisible := 'False'} : Bool := FALSE;   // I162.5
      "I162.6" { ExternalVisible := 'False'} : Bool := FALSE;   // I162.6
      "I162.7" { ExternalVisible := 'False'} : Bool := FALSE;   // I162.7
      "I163.0" { ExternalVisible := 'False'} : Bool := FALSE;   // I163.0
      "I163.1" { ExternalVisible := 'False'} : Bool := FALSE;   // I163.1
      "I163.2" { ExternalVisible := 'False'} : Bool := FALSE;   // I163.2
      "I163.3" { ExternalVisible := 'False'} : Bool := FALSE;   // I163.3
      "I163.4" { ExternalVisible := 'False'} : Bool := FALSE;   // I163.4
      "I163.5" { ExternalVisible := 'False'} : Bool := FALSE;   // I163.5
      "I163.6" { ExternalVisible := 'False'} : Bool := FALSE;   // I163.6
      "I163.7" { ExternalVisible := 'False'} : Bool := FALSE;   // I163.7
      "I164.0" { ExternalVisible := 'False'} : Bool := FALSE;   // I164.0
      "I164.1" { ExternalVisible := 'False'} : Bool := FALSE;   // I164.1
      "I164.2" { ExternalVisible := 'False'} : Bool := FALSE;   // I164.2
      "I164.3" { ExternalVisible := 'False'} : Bool := FALSE;   // I164.3
      "I164.4" { ExternalVisible := 'False'} : Bool := FALSE;   // I164.4
      "I164.5" { ExternalVisible := 'False'} : Bool := FALSE;   // I164.5
      "I164.6" { ExternalVisible := 'False'} : Bool := FALSE;   // I164.6
      "I164.7" { ExternalVisible := 'False'} : Bool := FALSE;   // I164.7
      "I165.0" { ExternalVisible := 'False'} : Bool := FALSE;   // I165.0
      "I165.1" { ExternalVisible := 'False'} : Bool := FALSE;   // I165.1
      "I165.2" { ExternalVisible := 'False'} : Bool := FALSE;   // I165.2
      "I165.3" { ExternalVisible := 'False'} : Bool := FALSE;   // I165.3
      "I165.4" { ExternalVisible := 'False'} : Bool := FALSE;   // I165.4
      "I165.5" { ExternalVisible := 'False'} : Bool := FALSE;   // I165.5
      "I165.6" { ExternalVisible := 'False'} : Bool := FALSE;   // I165.6
      "I165.7" { ExternalVisible := 'False'} : Bool := FALSE;   // I165.7
      "I166.0" { ExternalVisible := 'False'} : Bool := FALSE;   // I166.0
      "I166.1" { ExternalVisible := 'False'} : Bool := FALSE;   // I166.1
      "I166.2" { ExternalVisible := 'False'} : Bool := FALSE;   // I166.2
      "I166.3" { ExternalVisible := 'False'} : Bool := FALSE;   // I166.3
      "I166.4" { ExternalVisible := 'False'} : Bool := FALSE;   // I166.4
      "I166.5" { ExternalVisible := 'False'} : Bool := FALSE;   // I166.5
      "I166.6" { ExternalVisible := 'False'} : Bool := FALSE;   // I166.6
      "I166.7" { ExternalVisible := 'False'} : Bool := FALSE;   // I166.7
      "I167.0" { ExternalVisible := 'False'} : Bool := FALSE;   // I167.0
      "I167.1" { ExternalVisible := 'False'} : Bool := FALSE;   // I167.1
      "I167.2" { ExternalVisible := 'False'} : Bool := FALSE;   // I167.2
      "I167.3" { ExternalVisible := 'False'} : Bool := FALSE;   // I167.3
      "I167.4" { ExternalVisible := 'False'} : Bool := FALSE;   // I167.4
      "I167.5" { ExternalVisible := 'False'} : Bool := FALSE;   // I167.5
      "I167.6" { ExternalVisible := 'False'} : Bool := FALSE;   // I167.6
      "I167.7" { ExternalVisible := 'False'} : Bool := FALSE;   // I167.7
      "I168.0" { ExternalVisible := 'False'} : Bool := FALSE;   // I168.0
      "I168.1" { ExternalVisible := 'False'} : Bool := FALSE;   // I168.1
      "I168.2" { ExternalVisible := 'False'} : Bool := FALSE;   // I168.2
      "I168.3" { ExternalVisible := 'False'} : Bool := FALSE;   // I168.3
      "I168.4" { ExternalVisible := 'False'} : Bool := FALSE;   // I168.4
      "I168.5" { ExternalVisible := 'False'} : Bool := FALSE;   // I168.5
      "I168.6" { ExternalVisible := 'False'} : Bool := FALSE;   // I168.6
      "I168.7" { ExternalVisible := 'False'} : Bool := FALSE;   // I168.7
      "I169.0" { ExternalVisible := 'False'} : Bool := FALSE;   // I169.0
      "I169.1" { ExternalVisible := 'False'} : Bool := FALSE;   // I169.1
      "I169.2" { ExternalVisible := 'False'} : Bool := FALSE;   // I169.2
      "I169.3" { ExternalVisible := 'False'} : Bool := FALSE;   // I169.3
      "I169.4" { ExternalVisible := 'False'} : Bool := FALSE;   // I169.4
      "I169.5" { ExternalVisible := 'False'} : Bool := FALSE;   // I169.5
      "I169.6" { ExternalVisible := 'False'} : Bool := FALSE;   // I169.6
      "I169.7" { ExternalVisible := 'False'} : Bool := FALSE;   // I169.7
      "I170.0" { ExternalVisible := 'False'} : Bool := FALSE;   // I170.0
      "I170.1" { ExternalVisible := 'False'} : Bool := FALSE;   // I170.1
      "I170.2" { ExternalVisible := 'False'} : Bool := FALSE;   // I170.2
      "I170.3" { ExternalVisible := 'False'} : Bool := FALSE;   // I170.3
      "I170.4" { ExternalVisible := 'False'} : Bool := FALSE;   // I170.4
      "I170.5" { ExternalVisible := 'False'} : Bool := FALSE;   // I170.5
      "I170.6" { ExternalVisible := 'False'} : Bool := FALSE;   // I170.6
      "I170.7" { ExternalVisible := 'False'} : Bool := FALSE;   // I170.7
      "I171.0" { ExternalVisible := 'False'} : Bool := FALSE;   // I171.0
      "I171.1" { ExternalVisible := 'False'} : Bool := FALSE;   // I171.1
      "I171.2" { ExternalVisible := 'False'} : Bool := FALSE;   // I171.2
      "I171.3" { ExternalVisible := 'False'} : Bool := FALSE;   // I171.3
